C09095=1086.401,201.775,-73.711,175.633,21.629,153.454
C09096=1086.407,202.025,-73.734,175.636,21.631,153.454
C09097=1086.413,202.273,-73.758,175.638,21.633,153.454
C09098=1086.418,202.522,-73.781,175.641,21.634,153.454
C09099=1086.424,202.770,-73.805,175.644,21.636,153.454
C09100=1086.429,203.020,-73.828,175.647,21.638,153.453
C09101=1086.436,203.268,-73.852,175.649,21.640,153.454
C09102=1086.441,203.517,-73.876,175.652,21.641,153.453
C09103=1086.446,203.766,-73.900,175.654,21.643,153.453
C09104=1086.452,204.015,-73.923,175.657,21.644,153.453
C09105=1086.457,204.264,-73.947,175.659,21.646,153.453
C09106=1086.463,204.512,-73.971,175.663,21.648,153.453
C09107=1086.468,204.761,-73.995,175.665,21.650,153.453
C09108=1086.474,205.010,-74.019,175.668,21.651,153.453
C09109=1086.480,205.258,-74.042,175.670,21.653,153.453
C09110=1086.485,205.507,-74.066,175.673,21.654,153.453
C09111=1086.491,205.756,-74.090,175.675,21.656,153.453
C09112=1086.497,206.005,-74.114,175.679,21.658,153.453
C09113=1086.502,206.254,-74.138,175.681,21.660,153.453
C09114=1086.508,206.502,-74.161,175.684,21.661,153.453
C09115=1086.513,206.751,-74.186,175.686,21.663,153.453
C09116=1086.519,207.001,-74.210,175.689,21.665,153.453
C09117=1086.525,207.249,-74.233,175.692,21.666,153.453
C09118=1086.547,208.275,-74.332,175.771,21.707,153.449
C09119=1086.557,208.662,-74.370,175.775,21.711,153.449
C09120=1086.565,209.049,-74.408,175.779,21.715,153.450
C09121=1086.574,209.435,-74.446,175.782,21.719,153.450
C09122=1086.582,209.821,-74.484,175.787,21.723,153.450
C09123=1086.588,210.071,-74.509,175.789,21.726,153.450
C09124=1086.594,210.319,-74.532,175.792,21.728,153.450
C09125=1086.600,210.568,-74.557,175.795,21.731,153.451
C09126=1086.605,210.816,-74.582,175.797,21.733,153.451
C09127=1086.611,211.065,-74.606,175.800,21.736,153.451
C09128=1086.617,211.314,-74.631,175.802,21.738,153.451
C09129=1086.622,211.563,-74.655,175.805,21.741,153.451
C09130=1086.628,211.812,-74.680,175.807,21.744,153.451
C09131=1086.633,212.060,-74.705,175.810,21.747,153.452
C09132=1086.639,212.309,-74.729,175.813,21.749,153.452
C09133=1086.645,212.558,-74.754,175.815,21.752,153.452
C09134=1086.650,212.806,-74.779,175.818,21.754,153.452
C09135=1086.656,213.055,-74.803,175.820,21.757,153.452
C09136=1086.661,213.304,-74.827,175.823,21.760,153.452
C09137=1086.667,213.553,-74.852,175.825,21.762,153.453
C09138=1086.672,213.801,-74.878,175.829,21.765,153.453
C09139=1086.678,214.051,-74.902,175.831,21.767,153.453
C09140=1086.683,214.299,-74.926,175.833,21.770,153.453
C09141=1086.689,214.547,-74.951,175.836,21.772,153.453
C09142=1086.695,214.796,-74.976,175.838,21.775,153.453
C09143=1086.700,215.044,-75.001,175.841,21.778,153.454
C09144=1086.706,215.294,-75.026,175.843,21.780,153.454
C09145=1086.711,215.543,-75.051,175.847,21.783,153.454
C09146=1086.717,215.791,-75.076,175.849,21.786,153.454
C09147=1086.722,216.040,-75.100,175.852,21.788,153.454
C09148=1086.729,216.288,-75.125,175.854,21.791,153.454
C09149=1086.734,216.537,-75.150,175.856,21.793,153.454
C09150=1086.740,216.786,-75.175,175.859,21.796,153.455
C09151=1086.745,217.035,-75.200,175.862,21.798,153.455
C09152=1086.751,217.283,-75.225,175.865,21.801,153.455
C09153=1086.756,217.532,-75.249,175.867,21.804,153.455
C09154=1086.762,217.781,-75.275,175.870,21.806,153.455
C09155=1086.768,218.029,-75.299,175.872,21.809,153.456
C09156=1086.773,218.278,-75.325,175.875,21.812,153.456
C09157=1086.779,218.527,-75.350,175.877,21.814,153.456
C09158=1086.785,218.775,-75.375,175.881,21.817,153.456
C09159=1086.791,219.025,-75.399,175.883,21.820,153.456
C09160=1086.795,219.273,-75.425,175.886,21.822,153.456
C09161=1086.802,219.522,-75.450,175.888,21.825,153.456
C09162=1086.807,219.770,-75.474,175.891,21.828,153.457
C09163=1086.813,220.019,-75.500,175.893,21.830,153.457
C09164=1086.818,220.268,-75.525,175.896,21.832,153.457
C09165=1086.824,220.516,-75.550,175.899,21.835,153.457
C09166=1086.830,220.765,-75.575,175.901,21.837,153.457
C09167=1086.836,221.014,-75.600,175.904,21.840,153.457
C09168=1086.841,221.263,-75.625,175.906,21.843,153.457
C09169=1086.847,221.511,-75.651,175.909,21.845,153.458
C09170=1086.853,221.759,-75.676,175.912,21.848,153.458
C09171=1086.862,222.150,-75.715,175.916,21.852,153.458
C09172=1086.870,222.541,-75.755,175.920,21.856,153.458
C09173=1086.879,222.931,-75.794,175.925,21.861,153.459
C09174=1086.887,223.322,-75.835,175.928,21.865,153.459
C09175=1086.894,223.570,-75.860,175.931,21.868,153.459
C09176=1086.899,223.818,-75.885,175.934,21.870,153.459
C09177=1086.904,224.068,-75.910,175.937,21.873,153.459
C09178=1086.910,224.317,-75.936,175.939,21.875,153.460
C09179=1086.916,224.565,-75.961,175.942,21.878,153.460
C09180=1086.921,224.814,-75.987,175.944,21.880,153.460
C09181=1086.927,225.062,-76.012,175.947,21.883,153.460
C09182=1086.932,225.311,-76.038,175.950,21.885,153.460
C09183=1086.938,225.559,-76.063,175.952,21.889,153.460
C09184=1086.944,225.808,-76.089,175.955,21.891,153.461
C09185=1086.949,226.056,-76.114,175.958,21.894,153.461
C09186=1086.955,226.305,-76.140,175.960,21.896,153.461
C09187=1086.961,226.554,-76.165,175.963,21.899,153.461
C09188=1086.966,226.804,-76.191,175.965,21.901,153.461
C09189=1086.972,227.051,-76.216,175.968,21.904,153.461
C09190=1086.977,227.300,-76.241,175.972,21.907,153.461
C09191=1086.983,227.549,-76.267,175.974,21.909,153.462
C09192=1086.989,227.797,-76.293,175.977,21.912,153.462
C09193=1086.995,228.045,-76.318,175.979,21.915,153.462
C09194=1087.000,228.294,-76.344,175.982,21.917,153.462
C09195=1087.007,228.543,-76.370,175.985,21.920,153.462
C09196=1087.012,228.792,-76.396,175.987,21.923,153.462
C09197=1087.017,229.040,-76.421,175.990,21.925,153.463
C09198=1087.023,229.289,-76.446,175.993,21.928,153.463
C09199=1087.029,229.538,-76.472,175.995,21.931,153.463
C09200=1087.035,229.787,-76.498,175.998,21.933,153.463
C09201=1087.040,230.036,-76.524,176.000,21.936,153.463
C09202=1087.046,230.284,-76.549,176.003,21.939,153.463
C09203=1087.052,230.532,-76.575,176.006,21.941,153.464
C09204=1087.057,230.781,-76.601,176.009,21.944,153.464
C09205=1087.063,231.030,-76.627,176.012,21.947,153.464
C09206=1087.068,231.278,-76.652,176.014,21.949,153.464
C09207=1087.074,231.527,-76.678,176.017,21.952,153.464
C09208=1087.079,231.775,-76.705,176.019,21.955,153.464
C09209=1087.085,232.024,-76.731,176.022,21.957,153.465
C09210=1087.091,232.273,-76.756,176.025,21.960,153.465
C09211=1087.096,232.522,-76.782,176.028,21.963,153.465
C09212=1087.102,232.770,-76.808,176.030,21.965,153.465
C09213=1087.107,233.019,-76.834,176.033,21.968,153.465
C09214=1087.113,233.267,-76.859,176.036,21.971,153.465
C09215=1087.119,233.516,-76.886,176.038,21.973,153.466
C09216=1087.125,233.765,-76.912,176.041,21.976,153.466
C09217=1087.130,234.014,-76.938,176.044,21.978,153.466
C09218=1087.135,234.261,-76.964,176.047,21.981,153.466
C09219=1087.141,234.510,-76.990,176.049,21.984,153.466
C09220=1087.147,234.759,-77.016,176.052,21.986,153.466
C09221=1087.153,235.007,-77.042,176.055,21.990,153.467
C09222=1087.158,235.256,-77.068,176.057,21.992,153.467
C09223=1087.166,235.637,-77.108,176.062,21.996,153.467
C09224=1087.175,236.019,-77.149,176.066,22.000,153.467
C09225=1087.184,236.402,-77.188,176.070,22.005,153.468
C09226=1087.192,236.783,-77.228,176.074,22.009,153.468
C09227=1087.198,237.031,-77.255,176.077,22.011,153.468
C09228=1087.204,237.280,-77.281,176.079,22.014,153.468
C09229=1087.209,237.529,-77.307,176.082,22.017,153.468
C09230=1087.215,237.778,-77.333,176.085,22.019,153.469
C09231=1087.221,238.026,-77.360,176.088,22.022,153.469
C09232=1087.226,238.274,-77.387,176.091,22.025,153.469
C09233=1087.232,238.523,-77.413,176.093,22.027,153.469
C09234=1087.238,238.772,-77.439,176.096,22.030,153.469
C09235=1087.243,239.021,-77.465,176.098,22.032,153.469
C09236=1087.249,239.269,-77.492,176.101,22.036,153.470
C09237=1087.255,239.517,-77.519,176.104,22.038,153.470
C09238=1087.260,239.766,-77.544,176.107,22.041,153.470
C09239=1087.266,240.015,-77.571,176.110,22.044,153.470
C09240=1087.272,240.263,-77.598,176.112,22.046,153.470
C09241=1087.277,240.512,-77.624,176.115,22.049,153.470
C09242=1087.283,240.761,-77.650,176.118,22.052,153.471
C09243=1087.289,241.009,-77.677,176.120,22.054,153.471
C09244=1087.294,241.258,-77.703,176.124,22.057,153.471
C09245=1087.300,241.506,-77.730,176.127,22.060,153.471
C09246=1087.306,241.755,-77.756,176.129,22.062,153.471
C09247=1087.312,242.003,-77.783,176.132,22.065,153.471
C09248=1087.317,242.252,-77.809,176.134,22.068,153.472
C09249=1087.323,242.500,-77.835,176.137,22.070,153.472
C09250=1087.329,242.749,-77.862,176.140,22.074,153.472
C09251=1087.334,242.997,-77.889,176.143,22.076,153.472
C09252=1087.340,243.245,-77.915,176.146,22.079,153.472
C09253=1087.345,243.495,-77.942,176.148,22.081,153.473
C09254=1087.351,243.743,-77.969,176.151,22.084,153.473
C09255=1087.356,243.991,-77.995,176.154,22.087,153.473
C09256=1087.362,244.240,-78.022,176.156,22.090,153.473
C09257=1087.367,244.488,-78.049,176.159,22.092,153.473
C09258=1087.373,244.737,-78.076,176.162,22.095,153.473
C09259=1087.379,244.985,-78.102,176.164,22.098,153.474
C09260=1087.384,245.233,-78.129,176.168,22.101,153.474
C09261=1087.390,245.482,-78.156,176.171,22.104,153.474
C09262=1087.396,245.731,-78.183,176.173,22.106,153.474
C09263=1087.402,245.980,-78.210,176.176,22.109,153.474
C09264=1087.407,246.229,-78.236,176.179,22.112,153.475
C09265=1087.412,246.477,-78.263,176.181,22.114,153.475
C09266=1087.418,246.725,-78.290,176.184,22.117,153.475
C09267=1087.424,246.973,-78.317,176.187,22.119,153.475
C09268=1087.430,247.222,-78.344,176.190,22.123,153.475
C09269=1087.435,247.470,-78.371,176.193,22.125,153.476
C09270=1087.441,247.719,-78.398,176.195,22.128,153.476
C09271=1087.446,247.967,-78.425,176.198,22.131,153.476
C09272=1087.451,248.216,-78.452,176.201,22.134,153.476
C09273=1087.457,248.465,-78.479,176.203,22.136,153.476
C09274=1087.463,248.713,-78.506,176.206,22.139,153.476
C09275=1087.472,249.088,-78.547,176.211,22.144,153.477
C09276=1087.479,249.463,-78.587,176.215,22.147,153.477
C09277=1087.488,249.837,-78.628,176.219,22.152,153.477
C09278=1087.496,250.213,-78.669,176.223,22.156,153.478
C09279=1087.501,250.462,-78.696,176.226,22.159,153.478
C09280=1087.507,250.709,-78.724,176.229,22.162,153.478
C09281=1087.514,250.958,-78.751,176.231,22.164,153.478
C09282=1087.519,251.207,-78.778,176.234,22.168,153.478
C09283=1087.524,251.456,-78.805,176.237,22.170,153.479
C09284=1087.530,251.704,-78.832,176.240,22.173,153.479
C09285=1087.535,251.952,-78.860,176.243,22.176,153.479
C09286=1087.540,252.201,-78.886,176.246,22.179,153.479
C09287=1087.546,252.449,-78.915,176.248,22.181,153.479
C09288=1087.552,252.698,-78.941,176.251,22.184,153.480
C09289=1087.557,252.946,-78.969,176.254,22.187,153.480
C09290=1087.563,253.194,-78.996,176.256,22.189,153.480
C09291=1087.569,253.444,-79.024,176.259,22.192,153.480
C09292=1087.575,253.692,-79.050,176.262,22.196,153.480
C09293=1087.580,253.940,-79.078,176.266,22.198,153.481
C09294=1087.586,254.188,-79.105,176.268,22.201,153.481
C09295=1087.591,254.436,-79.133,176.271,22.204,153.481
C09296=1087.597,254.686,-79.160,176.274,22.207,153.481
C09297=1087.603,254.934,-79.187,176.276,22.209,153.481
C09298=1087.608,255.182,-79.215,176.279,22.212,153.482
C09299=1087.614,255.431,-79.242,176.282,22.215,153.482
C09300=1087.620,255.679,-79.270,176.284,22.217,153.482
C09301=1087.625,255.928,-79.297,176.288,22.220,153.482
C09302=1087.631,256.176,-79.325,176.291,22.224,153.482
C09303=1087.637,256.424,-79.353,176.294,22.226,153.483
C09304=1087.642,256.673,-79.380,176.296,22.229,153.483
C09305=1087.648,256.921,-79.407,176.299,22.232,153.483
C09306=1087.653,257.170,-79.435,176.302,22.235,153.483
C09307=1087.660,257.418,-79.462,176.304,22.237,153.483
C09308=1087.665,257.667,-79.490,176.307,22.240,153.483
C09309=1087.671,257.915,-79.517,176.310,22.243,153.484
C09310=1087.677,258.163,-79.545,176.313,22.246,153.484
C09311=1087.682,258.412,-79.573,176.316,22.248,153.484
C09312=1087.688,258.660,-79.600,176.319,22.251,153.484
C09313=1087.694,258.908,-79.628,176.322,22.254,153.484
C09314=1087.699,259.158,-79.656,176.325,22.257,153.485
C09315=1087.705,259.405,-79.683,176.327,22.259,153.485
C09316=1087.711,259.653,-79.711,176.330,22.263,153.485
C09317=1087.716,259.903,-79.739,176.333,22.265,153.485
C09318=1087.722,260.150,-79.766,176.336,22.268,153.485
C09319=1087.728,260.399,-79.795,176.339,22.271,153.486
C09320=1087.734,260.647,-79.823,176.342,22.274,153.486
C09321=1087.740,260.895,-79.850,176.345,22.277,153.486
C09322=1087.745,261.144,-79.877,176.347,22.279,153.486
C09323=1087.751,261.392,-79.905,176.350,22.282,153.486
C09324=1087.757,261.641,-79.934,176.353,22.285,153.487
C09325=1087.763,261.889,-79.961,176.356,22.288,153.487
C09326=1087.769,262.138,-79.989,176.358,22.290,153.487
C09327=1087.777,262.510,-80.031,176.363,22.295,153.487
C09328=1087.786,262.882,-80.073,176.368,22.299,153.487
C09329=1087.794,263.254,-80.115,176.371,22.303,153.488
C09330=1087.803,263.626,-80.156,176.376,22.307,153.488
C09331=1087.810,263.875,-80.184,176.379,22.310,153.488
C09332=1087.815,264.123,-80.212,176.381,22.312,153.488
C09333=1087.821,264.371,-80.240,176.384,22.316,153.489
C09334=1087.826,264.619,-80.268,176.388,22.318,153.489
C09335=1087.832,264.868,-80.297,176.390,22.322,153.489
C09336=1087.837,265.116,-80.325,176.394,22.324,153.489
C09337=1087.843,265.365,-80.353,176.396,22.327,153.490
C09338=1087.849,265.613,-80.381,176.399,22.330,153.490
C09339=1087.855,265.862,-80.409,176.402,22.333,153.490
C09340=1087.860,266.110,-80.437,176.405,22.336,153.490
C09341=1087.866,266.359,-80.466,176.407,22.338,153.490
C09342=1087.871,266.607,-80.493,176.410,22.342,153.491
C09343=1087.877,266.855,-80.521,176.413,22.344,153.491
C09344=1087.883,267.103,-80.550,176.416,22.348,153.491
C09345=1087.889,267.352,-80.579,176.419,22.350,153.491
C09346=1087.894,267.600,-80.607,176.421,22.353,153.492
C09347=1087.900,267.848,-80.635,176.425,22.356,153.492
C09348=1087.905,268.096,-80.663,176.428,22.359,153.492
C09349=1087.911,268.345,-80.691,176.431,22.362,153.492
C09350=1087.917,268.593,-80.720,176.433,22.364,153.492
C09351=1087.923,268.841,-80.748,176.436,22.368,153.493
C09352=1087.928,269.090,-80.777,176.439,22.370,153.493
C09353=1087.934,269.338,-80.805,176.442,22.374,153.493
C09354=1087.939,269.586,-80.834,176.445,22.377,153.493
C09355=1087.945,269.835,-80.862,176.447,22.379,153.493
C09356=1087.951,270.083,-80.891,176.450,22.382,153.494
C09357=1087.957,270.331,-80.919,176.453,22.385,153.494
C09358=1087.963,270.580,-80.948,176.456,22.388,153.494
C09359=1087.968,270.828,-80.976,176.459,22.391,153.494
C09360=1087.974,271.076,-81.005,176.463,22.394,153.495
C09361=1087.979,271.325,-81.033,176.465,22.397,153.495
C09362=1087.985,271.573,-81.061,176.468,22.400,153.495
C09363=1087.991,271.821,-81.090,176.471,22.403,153.495
C09364=1087.996,272.069,-81.118,176.474,22.406,153.495
C09365=1088.002,272.317,-81.148,176.477,22.409,153.496
C09366=1088.008,272.566,-81.176,176.479,22.411,153.496
C09367=1088.013,272.814,-81.204,176.482,22.415,153.496
C09368=1088.019,273.062,-81.233,176.485,22.417,153.496
C09369=1088.024,273.311,-81.262,176.488,22.421,153.497
C09370=1088.030,273.559,-81.291,176.491,22.423,153.497
C09371=1088.036,273.808,-81.319,176.494,22.427,153.497
C09372=1088.042,274.055,-81.348,176.497,22.429,153.497
C09373=1088.047,274.304,-81.377,176.500,22.432,153.498
C09374=1088.053,274.552,-81.406,176.502,22.435,153.498
C09375=1088.059,274.800,-81.435,176.506,22.438,153.498
C09376=1088.064,275.049,-81.464,176.509,22.441,153.498
C09377=1088.070,275.297,-81.493,176.512,22.444,153.498
C09378=1088.076,275.545,-81.521,176.514,22.447,153.499
C09379=1088.085,275.920,-81.564,176.518,22.452,153.499
C09380=1088.093,276.295,-81.608,176.523,22.456,153.499
C09381=1088.102,276.670,-81.652,176.527,22.461,153.500
C09382=1088.110,277.044,-81.696,176.532,22.466,153.500
C09383=1088.116,277.293,-81.724,176.534,22.468,153.500
C09384=1088.122,277.541,-81.754,176.537,22.471,153.501
C09385=1088.127,277.790,-81.783,176.540,22.474,153.501
C09386=1088.133,278.037,-81.812,176.543,22.477,153.501
C09387=1088.138,278.286,-81.841,176.546,22.480,153.501
C09388=1088.144,278.535,-81.870,176.549,22.483,153.502
C09389=1088.149,278.782,-81.899,176.552,22.486,153.502
C09390=1088.156,279.030,-81.928,176.554,22.489,153.502
C09391=1088.161,279.279,-81.958,176.558,22.492,153.502
C09392=1088.167,279.528,-81.986,176.561,22.495,153.503
C09393=1088.173,279.776,-82.016,176.564,22.498,153.503
C09394=1088.178,280.023,-82.044,176.567,22.501,153.503
C09395=1088.184,280.272,-82.074,176.570,22.504,153.503
C09396=1088.190,280.520,-82.103,176.573,22.508,153.504
C09397=1088.195,280.768,-82.133,176.576,22.510,153.504
C09398=1088.201,281.016,-82.161,176.578,22.513,153.504
C09399=1088.207,281.264,-82.191,176.581,22.516,153.504
C09400=1088.213,281.512,-82.220,176.584,22.519,153.505
C09401=1088.218,281.761,-82.250,176.587,22.523,153.505
C09402=1088.224,282.009,-82.279,176.590,22.526,153.505
C09403=1088.230,282.257,-82.308,176.593,22.529,153.505
C09404=1088.235,282.505,-82.338,176.596,22.532,153.506
C09405=1088.241,282.754,-82.367,176.599,22.535,153.506
C09406=1088.247,283.002,-82.396,176.602,22.538,153.506
C09407=1088.252,283.250,-82.426,176.604,22.541,153.506
C09408=1088.257,283.498,-82.455,176.607,22.544,153.507
C09409=1088.263,283.746,-82.484,176.610,22.547,153.507
C09410=1088.269,283.995,-82.514,176.613,22.550,153.507
C09411=1088.274,284.243,-82.543,176.616,22.554,153.507
C09412=1088.281,284.491,-82.573,176.619,22.557,153.508
C09413=1088.286,284.740,-82.602,176.622,22.560,153.508
C09414=1088.291,284.987,-82.631,176.625,22.563,153.508
C09415=1088.297,285.235,-82.662,176.628,22.566,153.508
C09416=1088.303,285.483,-82.691,176.631,22.569,153.509
C09417=1088.309,285.732,-82.720,176.634,22.572,153.509
C09418=1088.314,285.980,-82.750,176.636,22.575,153.509
C09419=1088.320,286.229,-82.780,176.639,22.578,153.510
C09420=1088.326,286.476,-82.809,176.642,22.581,153.510
C09421=1088.332,286.725,-82.839,176.645,22.585,153.510
C09422=1088.337,286.973,-82.869,176.649,22.587,153.510
C09423=1088.343,287.221,-82.898,176.652,22.591,153.511
C09424=1088.349,287.468,-82.928,176.655,22.594,153.511
C09425=1088.354,287.717,-82.957,176.657,22.597,153.511
C09426=1088.360,287.965,-82.987,176.660,22.600,153.511
C09427=1088.366,288.213,-83.017,176.664,22.603,153.512
C09428=1088.372,288.461,-83.046,176.667,22.606,153.512
C09429=1088.378,288.709,-83.077,176.670,22.609,153.512
C09430=1088.383,288.957,-83.106,176.673,22.613,153.512
C09431=1088.392,289.342,-83.152,176.677,22.617,153.513
C09432=1088.401,289.727,-83.199,176.681,22.622,153.513
C09433=1088.410,290.111,-83.245,176.686,22.627,153.514
C09434=1088.418,290.496,-83.292,176.690,22.632,153.514
C09435=1088.425,290.743,-83.321,176.693,22.635,153.515
C09436=1088.430,290.992,-83.351,176.696,22.639,153.515
C09437=1088.436,291.240,-83.381,176.699,22.642,153.515
C09438=1088.442,291.488,-83.411,176.703,22.645,153.515
C09439=1088.448,291.736,-83.441,176.705,22.648,153.516
C09440=1088.453,291.984,-83.471,176.708,22.651,153.516
C09441=1088.459,292.232,-83.501,176.711,22.654,153.516
C09442=1088.465,292.480,-83.532,176.714,22.657,153.516
C09443=1088.470,292.728,-83.561,176.717,22.661,153.517
C09444=1088.476,292.976,-83.592,176.720,22.664,153.517
C09445=1088.482,293.224,-83.622,176.723,22.667,153.517
C09446=1088.487,293.472,-83.652,176.726,22.670,153.518
C09447=1088.492,293.721,-83.683,176.729,22.674,153.518
C09448=1088.498,293.968,-83.713,176.732,22.677,153.518
C09449=1088.504,294.217,-83.743,176.734,22.680,153.519
C09450=1088.510,294.465,-83.773,176.737,22.683,153.519
C09451=1088.515,294.712,-83.803,176.740,22.686,153.519
C09452=1088.521,294.961,-83.833,176.743,22.689,153.519
C09453=1088.527,295.209,-83.863,176.746,22.693,153.520
C09454=1088.533,295.457,-83.894,176.749,22.696,153.520
C09455=1088.539,295.705,-83.924,176.752,22.699,153.520
C09456=1088.545,295.953,-83.955,176.755,22.702,153.521
C09457=1088.550,296.201,-83.984,176.758,22.705,153.521
C09458=1088.555,296.449,-84.015,176.761,22.709,153.521
C09459=1088.561,296.697,-84.046,176.764,22.712,153.522
C09460=1088.567,296.945,-84.076,176.767,22.716,153.522
C09461=1088.573,297.193,-84.106,176.770,22.719,153.522
C09462=1088.579,297.441,-84.137,176.773,22.722,153.522
C09463=1088.585,297.689,-84.167,176.776,22.725,153.523
C09464=1088.590,297.938,-84.198,176.779,22.728,153.523
C09465=1088.596,298.186,-84.228,176.782,22.732,153.523
C09466=1088.601,298.434,-84.258,176.785,22.735,153.524
C09467=1088.607,298.682,-84.289,176.789,22.739,153.524
C09468=1088.612,298.930,-84.320,176.792,22.742,153.524
C09469=1088.618,299.177,-84.350,176.795,22.746,153.525
C09470=1088.623,299.426,-84.381,176.797,22.749,153.525
C09471=1088.629,299.673,-84.411,176.800,22.752,153.525
C09472=1088.634,299.922,-84.442,176.803,22.756,153.526
C09473=1088.641,300.170,-84.473,176.806,22.759,153.526
C09474=1088.646,300.418,-84.504,176.809,22.763,153.526
C09475=1088.652,300.665,-84.535,176.812,22.766,153.527
C09476=1088.658,300.913,-84.565,176.815,22.769,153.527
C09477=1088.663,301.161,-84.596,176.818,22.773,153.527
C09478=1088.668,301.409,-84.627,176.821,22.776,153.528
C09479=1088.674,301.657,-84.658,176.824,22.779,153.528
C09480=1088.680,301.906,-84.688,176.827,22.783,153.528
C09481=1088.685,302.154,-84.719,176.830,22.786,153.529
C09482=1088.691,302.401,-84.750,176.833,22.789,153.529
C09483=1088.700,302.800,-84.800,176.838,22.795,153.530
C09484=1088.709,303.198,-84.849,176.842,22.800,153.530
C09485=1088.718,303.597,-84.899,176.848,22.806,153.531
C09486=1088.727,303.995,-84.949,176.852,22.811,153.531
C09487=1088.733,304.243,-84.979,176.855,22.815,153.532
C09488=1088.739,304.492,-85.011,176.858,22.818,153.532
C09489=1088.745,304.739,-85.042,176.861,22.822,153.532
C09490=1088.750,304.987,-85.073,176.864,22.825,153.533
C09491=1088.756,305.235,-85.103,176.867,22.829,153.533
C09492=1088.762,305.483,-85.135,176.870,22.832,153.533
C09493=1088.767,305.731,-85.166,176.873,22.835,153.534
C09494=1088.773,305.979,-85.196,176.876,22.839,153.534
C09495=1088.779,306.227,-85.229,176.879,22.842,153.534
C09496=1088.784,306.475,-85.259,176.882,22.846,153.535
C09497=1088.790,306.723,-85.291,176.885,22.849,153.535
C09498=1088.796,306.971,-85.321,176.888,22.852,153.535
C09499=1088.802,307.219,-85.353,176.891,22.856,153.536
C09500=1088.807,307.467,-85.383,176.894,22.859,153.536
C09501=1088.813,307.715,-85.415,176.897,22.863,153.537
C09502=1088.818,307.963,-85.446,176.900,22.867,153.537
C09503=1088.825,308.210,-85.477,176.903,22.870,153.537
C09504=1088.830,308.459,-85.509,176.906,22.873,153.538
C09505=1088.836,308.706,-85.540,176.909,22.877,153.538
C09506=1088.842,308.955,-85.571,176.912,22.880,153.538
C09507=1088.847,309.203,-85.603,176.915,22.884,153.539
C09508=1088.854,309.450,-85.634,176.918,22.887,153.539
C09509=1088.859,309.699,-85.665,176.921,22.890,153.539
C09510=1088.865,309.946,-85.697,176.924,22.894,153.540
C09511=1088.871,310.194,-85.728,176.928,22.898,153.540
C09512=1088.876,310.442,-85.759,176.930,22.901,153.540
C09513=1088.882,310.690,-85.791,176.933,22.905,153.541
C09514=1088.889,310.938,-85.822,176.936,22.908,153.541
C09515=1088.894,311.186,-85.853,176.939,22.912,153.542
C09516=1088.900,311.434,-85.885,176.942,22.915,153.542
C09517=1088.906,311.682,-85.917,176.945,22.918,153.542
C09518=1088.912,311.929,-85.948,176.948,22.922,153.543
C09519=1088.917,312.178,-85.980,176.951,22.925,153.543
C09520=1088.923,312.425,-86.011,176.955,22.929,153.543
C09521=1088.929,312.674,-86.043,176.958,22.933,153.544
C09522=1088.935,312.921,-86.074,176.960,22.936,153.544
C09523=1088.942,313.169,-86.106,176.964,22.940,153.544
C09524=1088.947,313.416,-86.137,176.966,22.943,153.545
C09525=1088.953,313.665,-86.169,176.969,22.946,153.545
C09526=1088.958,313.913,-86.200,176.972,22.950,153.546
C09527=1088.965,314.161,-86.232,176.976,22.954,153.546
C09528=1088.971,314.409,-86.264,176.979,22.957,153.546
C09529=1088.976,314.656,-86.295,176.982,22.961,153.547
C09530=1088.982,314.905,-86.327,176.985,22.964,153.547
C09531=1088.988,315.152,-86.359,176.988,22.968,153.547
C09532=1088.993,315.400,-86.391,176.990,22.972,153.548
C09533=1088.999,315.648,-86.423,176.993,22.975,153.548
C09534=1089.005,315.896,-86.455,176.997,22.979,153.549
C09535=1089.014,316.297,-86.507,177.001,22.985,153.549
C09536=1089.023,316.698,-86.558,177.006,22.991,153.550
C09537=1089.032,317.100,-86.610,177.011,22.997,153.551
C09538=1089.041,317.501,-86.662,177.016,23.003,153.551
C09539=1089.047,317.749,-86.693,177.019,23.007,153.552
C09540=1089.053,317.997,-86.725,177.022,23.011,153.552
C09541=1089.058,318.244,-86.757,177.025,23.014,153.553
C09542=1089.064,318.493,-86.789,177.028,23.018,153.553
C09543=1089.069,318.741,-86.822,177.031,23.022,153.554
C09544=1089.075,318.988,-86.854,177.034,23.026,153.554
C09545=1089.081,319.236,-86.886,177.037,23.029,153.554
C09546=1089.086,319.484,-86.918,177.040,23.033,153.555
C09547=1089.092,319.732,-86.950,177.043,23.037,153.555
C09548=1089.098,319.980,-86.983,177.046,23.040,153.556
C09549=1089.103,320.227,-87.015,177.049,23.044,153.556
C09550=1089.109,320.476,-87.047,177.052,23.048,153.557
C09551=1089.115,320.724,-87.079,177.055,23.052,153.557
C09552=1089.121,320.971,-87.111,177.058,23.055,153.558
C09553=1089.126,321.219,-87.144,177.061,23.059,153.558
C09554=1089.132,321.467,-87.176,177.064,23.063,153.558
C09555=1089.138,321.714,-87.208,177.067,23.067,153.559
C09556=1089.144,321.963,-87.240,177.070,23.071,153.559
C09557=1089.149,322.210,-87.274,177.073,23.074,153.560
C09558=1089.155,322.458,-87.305,177.076,23.078,153.560
C09559=1089.161,322.706,-87.337,177.080,23.082,153.561
C09560=1089.167,322.954,-87.370,177.082,23.086,153.561
C09561=1089.172,323.202,-87.403,177.085,23.089,153.561
C09562=1089.178,323.449,-87.435,177.088,23.093,153.562
C09563=1089.184,323.697,-87.467,177.092,23.098,153.562
C09564=1089.189,323.945,-87.500,177.095,23.101,153.563
C09565=1089.195,324.194,-87.532,177.097,23.105,153.563
C09566=1089.201,324.440,-87.565,177.100,23.109,153.564
C09567=1089.207,324.689,-87.597,177.103,23.112,153.564
C09568=1089.213,324.937,-87.630,177.107,23.116,153.565
C09569=1089.219,325.185,-87.662,177.109,23.120,153.565
C09570=1089.225,325.432,-87.695,177.112,23.124,153.566
C09571=1089.230,325.680,-87.727,177.115,23.128,153.566
C09572=1089.236,325.928,-87.760,177.119,23.132,153.566
C09573=1089.242,326.175,-87.793,177.122,23.136,153.567
C09574=1089.247,326.424,-87.825,177.124,23.140,153.567
C09575=1089.254,326.671,-87.858,177.127,23.143,153.568
C09576=1089.260,326.919,-87.891,177.131,23.147,153.568
C09577=1089.265,327.167,-87.923,177.134,23.151,153.569
C09578=1089.271,327.414,-87.956,177.137,23.155,153.569
C09579=1089.276,327.662,-87.989,177.139,23.159,153.570
C09580=1089.283,327.910,-88.022,177.143,23.163,153.570
C09581=1089.289,328.158,-88.054,177.146,23.167,153.571
C09582=1089.294,328.406,-88.087,177.149,23.170,153.571
C09583=1089.301,328.654,-88.120,177.152,23.175,153.572
C09584=1089.306,328.902,-88.153,177.155,23.178,153.572
C09585=1089.312,329.149,-88.186,177.158,23.182,153.572
C09586=1089.318,329.397,-88.218,177.161,23.186,153.573
C09587=1089.327,329.791,-88.271,177.166,23.193,153.574
C09588=1089.337,330.186,-88.323,177.171,23.199,153.574
C09589=1089.346,330.580,-88.376,177.176,23.205,153.575
C09590=1089.356,330.975,-88.428,177.181,23.211,153.576
C09591=1089.362,331.223,-88.461,177.184,23.215,153.577
C09592=1089.368,331.470,-88.494,177.186,23.219,153.577
C09593=1089.373,331.718,-88.527,177.190,23.223,153.577
C09594=1089.380,331.966,-88.560,177.193,23.227,153.578
C09595=1089.385,332.214,-88.593,177.196,23.231,153.578
C09596=1089.391,332.461,-88.627,177.199,23.235,153.579
C09597=1089.397,332.709,-88.659,177.202,23.240,153.580
C09598=1089.403,332.957,-88.693,177.205,23.243,153.580
C09599=1089.408,333.205,-88.726,177.208,23.248,153.581
C09600=1089.414,333.453,-88.760,177.211,23.252,153.581
C09601=1089.419,333.700,-88.792,177.214,23.256,153.582
C09602=1089.425,333.948,-88.825,177.218,23.260,153.582
C09603=1089.431,334.195,-88.859,177.220,23.264,153.583
C09604=1089.437,334.442,-88.892,177.223,23.268,153.583
C09605=1089.443,334.690,-88.925,177.227,23.272,153.584
C09606=1089.448,334.938,-88.959,177.229,23.277,153.584
C09607=1089.454,335.187,-88.992,177.232,23.281,153.585
C09608=1089.460,335.434,-89.026,177.236,23.285,153.585
C09609=1089.467,335.682,-89.059,177.239,23.289,153.586
C09610=1089.472,335.930,-89.093,177.242,23.293,153.586
C09611=1089.478,336.177,-89.126,177.245,23.297,153.587
C09612=1089.484,336.425,-89.160,177.248,23.302,153.588
C09613=1089.489,336.673,-89.193,177.251,23.306,153.588
C09614=1089.495,336.920,-89.226,177.254,23.310,153.589
C09615=1089.501,337.168,-89.260,177.257,23.314,153.589
C09616=1089.507,337.415,-89.293,177.260,23.318,153.590
C09617=1089.512,337.663,-89.327,177.263,23.323,153.590
C09618=1089.518,337.911,-89.361,177.267,23.327,153.591
C09619=1089.524,338.159,-89.394,177.269,23.331,153.591
C09620=1089.531,338.406,-89.428,177.272,23.335,153.592
C09621=1089.537,338.654,-89.461,177.276,23.339,153.592
C09622=1089.542,338.902,-89.495,177.278,23.343,153.593
C09623=1089.548,339.149,-89.529,177.282,23.348,153.593
C09624=1089.554,339.397,-89.562,177.285,23.352,153.594
C09625=1089.559,339.645,-89.596,177.287,23.357,153.595
C09626=1089.565,339.892,-89.629,177.291,23.361,153.595
C09627=1089.571,340.140,-89.663,177.294,23.365,153.596
C09628=1089.577,340.387,-89.698,177.297,23.370,153.596
C09629=1089.583,340.636,-89.731,177.300,23.374,153.597
C09630=1089.589,340.883,-89.765,177.303,23.378,153.598
C09631=1089.594,341.131,-89.799,177.306,23.383,153.598
C09632=1089.600,341.378,-89.833,177.309,23.387,153.599
C09633=1089.605,341.626,-89.867,177.312,23.391,153.599
C09634=1089.611,341.874,-89.901,177.315,23.396,153.600
C09635=1089.617,342.122,-89.935,177.319,23.400,153.601
C09636=1089.623,342.369,-89.969,177.321,23.404,153.601
C09637=1089.629,342.617,-90.002,177.325,23.409,153.602
C09638=1089.635,342.864,-90.036,177.328,23.413,153.602
C09639=1089.644,343.253,-90.090,177.332,23.420,153.603
C09640=1089.653,343.641,-90.143,177.337,23.427,153.604
C09641=1089.662,344.030,-90.197,177.342,23.434,153.605
C09642=1089.671,344.419,-90.251,177.347,23.441,153.606
C09643=1089.677,344.666,-90.285,177.349,23.445,153.607
C09644=1089.683,344.913,-90.319,177.353,23.450,153.607
C09645=1089.689,345.161,-90.353,177.356,23.454,153.608
C09646=1089.695,345.409,-90.386,177.359,23.459,153.609
C09647=1089.700,345.657,-90.421,177.362,23.463,153.609
C09648=1089.706,345.904,-90.455,177.365,23.468,153.610
C09649=1089.712,346.152,-90.490,177.368,23.472,153.610
C09650=1089.718,346.399,-90.524,177.371,23.477,153.611
C09651=1089.723,346.647,-90.558,177.374,23.481,153.612
C09652=1089.729,346.894,-90.592,177.378,23.486,153.612
C09653=1089.736,347.142,-90.627,177.380,23.491,153.613
C09654=1089.741,347.390,-90.661,177.384,23.495,153.614
C09655=1089.747,347.637,-90.695,177.386,23.500,153.614
C09656=1089.753,347.885,-90.730,177.390,23.504,153.615
C09657=1089.758,348.132,-90.765,177.393,23.509,153.616
C09658=1089.765,348.379,-90.799,177.396,23.514,153.616
C09659=1089.771,348.627,-90.834,177.399,23.518,153.617
C09660=1089.776,348.875,-90.868,177.402,23.523,153.618
C09661=1089.782,349.122,-90.902,177.405,23.527,153.618
C09662=1089.788,349.370,-90.937,177.408,23.532,153.619
C09663=1089.794,349.618,-90.971,177.411,23.537,153.620
C09664=1089.800,349.864,-91.006,177.414,23.542,153.620
C09665=1089.805,350.113,-91.041,177.417,23.546,153.621
C09666=1089.811,350.360,-91.075,177.421,23.551,153.622
C09667=1089.818,350.608,-91.110,177.424,23.556,153.622
C09668=1089.823,350.855,-91.145,177.427,23.560,153.623
C09669=1089.829,351.102,-91.179,177.430,23.565,153.624
C09670=1089.835,351.350,-91.214,177.433,23.570,153.624
C09671=1089.841,351.598,-91.248,177.436,23.575,153.625
C09672=1089.847,351.845,-91.284,177.439,23.579,153.626
C09673=1089.853,352.093,-91.318,177.442,23.584,153.626
C09674=1089.858,352.340,-91.353,177.445,23.588,153.627
C09675=1089.864,352.588,-91.388,177.448,23.593,153.628
C09676=1089.870,352.835,-91.422,177.452,23.598,153.628
C09677=1089.876,353.083,-91.458,177.454,23.603,153.629
C09678=1089.881,353.330,-91.492,177.458,23.608,153.630
C09679=1089.888,353.577,-91.527,177.460,23.612,153.631
C09680=1089.893,353.825,-91.562,177.464,23.617,153.631
C09681=1089.900,354.072,-91.597,177.466,23.622,153.632
C09682=1089.905,354.320,-91.632,177.470,23.627,153.633
C09683=1089.911,354.568,-91.667,177.473,23.632,153.633
C09684=1089.917,354.815,-91.702,177.476,23.637,153.634
C09685=1089.923,355.062,-91.737,177.479,23.642,153.635
C09686=1089.928,355.310,-91.772,177.482,23.646,153.636
C09687=1089.934,355.557,-91.807,177.485,23.651,153.636
C09688=1089.940,355.805,-91.842,177.488,23.657,153.637
C09689=1089.946,356.052,-91.877,177.491,23.661,153.638
C09690=1089.952,356.300,-91.912,177.494,23.666,153.638
C09691=1089.961,356.691,-91.968,177.499,23.674,153.640
C09692=1089.971,357.083,-92.024,177.504,23.681,153.641
C09693=1089.980,357.473,-92.080,177.509,23.690,153.642
C09694=1089.990,357.864,-92.135,177.514,23.697,153.643
C09695=1089.995,358.111,-92.170,177.517,23.703,153.644
C09696=1090.001,358.360,-92.205,177.520,23.707,153.645
C09697=1090.006,358.607,-92.241,177.523,23.713,153.646
C09698=1090.013,358.854,-92.276,177.526,23.718,153.646
C09699=1090.019,359.102,-92.312,177.529,23.723,153.647
C09700=1090.025,359.349,-92.347,177.532,23.728,153.648
C09701=1090.031,359.596,-92.383,177.536,23.733,153.649
C09702=1090.037,359.843,-92.418,177.538,23.737,153.649
C09703=1090.043,360.091,-92.453,177.542,23.743,153.650
C09704=1090.049,360.339,-92.488,177.545,23.748,153.651
C09705=1090.054,360.586,-92.524,177.547,23.753,153.652
C09706=1090.060,360.834,-92.559,177.551,23.758,153.653
C09707=1090.065,361.081,-92.595,177.554,23.764,153.653
C09708=1090.071,361.328,-92.630,177.557,23.768,153.654
C09709=1090.078,361.575,-92.667,177.560,23.774,153.655
C09710=1090.083,361.822,-92.702,177.563,23.779,153.656
C09711=1090.090,362.070,-92.737,177.566,23.784,153.657
C09712=1090.096,362.317,-92.773,177.569,23.789,153.657
C09713=1090.101,362.564,-92.809,177.573,23.794,153.658
C09714=1090.108,362.812,-92.844,177.575,23.799,153.659
C09715=1090.114,363.060,-92.880,177.578,23.805,153.660
C09716=1090.119,363.307,-92.915,177.582,23.810,153.661
C09717=1090.125,363.554,-92.952,177.585,23.816,153.661
C09718=1090.131,363.801,-92.988,177.587,23.821,153.662
C09719=1090.137,364.049,-93.023,177.591,23.826,153.663
C09720=1090.143,364.296,-93.059,177.594,23.831,153.664
C09721=1090.149,364.544,-93.094,177.596,23.836,153.665
C09722=1090.155,364.791,-93.131,177.600,23.842,153.666
C09723=1090.161,365.038,-93.166,177.603,23.847,153.666
C09724=1090.167,365.285,-93.202,177.606,23.853,153.667
C09725=1090.173,365.533,-93.238,177.609,23.857,153.668
C09726=1090.179,365.780,-93.274,177.612,23.863,153.669
C09727=1090.184,366.027,-93.310,177.616,23.868,153.670
C09728=1090.190,366.275,-93.346,177.619,23.874,153.671
C09729=1090.196,366.522,-93.382,177.621,23.879,153.672
C09730=1090.202,366.769,-93.419,177.625,23.885,153.672
C09731=1090.208,367.016,-93.454,177.628,23.890,153.673
C09732=1090.213,367.264,-93.491,177.631,23.896,153.674
C09733=1090.219,367.511,-93.527,177.634,23.901,153.675
C09734=1090.225,367.759,-93.562,177.637,23.907,153.676
C09735=1090.231,368.005,-93.599,177.640,23.912,153.677
C09736=1090.238,368.252,-93.635,177.643,23.918,153.678
C09737=1090.243,368.500,-93.671,177.646,23.923,153.679
C09738=1090.249,368.747,-93.708,177.649,23.929,153.680
C09739=1090.255,368.995,-93.744,177.652,23.934,153.680
C09740=1090.260,369.242,-93.780,177.655,23.940,153.681
C09741=1090.267,369.489,-93.817,177.658,23.945,153.682
C09742=1090.273,369.736,-93.852,177.661,23.951,153.683
C09743=1090.282,370.143,-93.912,177.666,23.960,153.685
C09744=1090.291,370.550,-93.972,177.671,23.969,153.686
C09745=1090.302,370.956,-94.032,177.676,23.979,153.688
C09746=1090.312,371.363,-94.092,177.682,23.988,153.689
C09747=1090.318,371.610,-94.128,177.685,23.993,153.690
C09748=1090.323,371.858,-94.165,177.688,23.999,153.691
C09749=1090.330,372.105,-94.201,177.690,24.005,153.692
C09750=1090.336,372.352,-94.238,177.694,24.011,153.693
C09751=1090.342,372.599,-94.275,177.697,24.016,153.694
C09752=1090.348,372.846,-94.311,177.700,24.022,153.695
C09753=1090.354,373.093,-94.347,177.703,24.028,153.696
C09754=1090.359,373.340,-94.384,177.707,24.033,153.697
C09755=1090.366,373.587,-94.421,177.709,24.039,153.698
C09756=1090.371,373.835,-94.457,177.712,24.045,153.699
C09757=1090.377,374.082,-94.493,177.715,24.051,153.700
C09758=1090.383,374.330,-94.531,177.719,24.056,153.701
C09759=1090.389,374.577,-94.567,177.722,24.062,153.702
C09760=1090.395,374.824,-94.604,177.725,24.068,153.703
C09761=1090.402,375.070,-94.641,177.728,24.074,153.704
C09762=1090.407,375.318,-94.678,177.730,24.080,153.705
C09763=1090.414,375.565,-94.715,177.733,24.086,153.706
C09764=1090.419,375.812,-94.752,177.737,24.092,153.707
C09765=1090.425,376.060,-94.789,177.740,24.098,153.708
C09766=1090.431,376.307,-94.825,177.743,24.104,153.709
C09767=1090.437,376.554,-94.862,177.746,24.110,153.710
C09768=1090.443,376.801,-94.899,177.749,24.116,153.711
C09769=1090.449,377.048,-94.936,177.752,24.122,153.712
C09770=1090.454,377.295,-94.973,177.756,24.128,153.713
C09771=1090.461,377.542,-95.010,177.758,24.134,153.714
C09772=1090.466,377.790,-95.047,177.761,24.139,153.715
C09773=1090.472,378.036,-95.085,177.764,24.146,153.716
C09774=1090.479,378.283,-95.121,177.767,24.152,153.717
C09775=1090.484,378.531,-95.158,177.770,24.158,153.718
C09776=1090.490,378.777,-95.196,177.774,24.164,153.719
C09777=1090.497,379.025,-95.232,177.777,24.170,153.720
C09778=1090.502,379.272,-95.269,177.780,24.176,153.721
C09779=1090.508,379.519,-95.307,177.783,24.182,153.722
C09780=1090.514,379.766,-95.344,177.786,24.189,153.723
C09781=1090.521,380.013,-95.382,177.789,24.195,153.724
C09782=1090.526,380.261,-95.419,177.792,24.201,153.725
C09783=1090.533,380.507,-95.456,177.795,24.207,153.726
C09784=1090.539,380.754,-95.493,177.799,24.213,153.728
C09785=1090.545,381.001,-95.531,177.802,24.220,153.729
C09786=1090.550,381.248,-95.568,177.805,24.226,153.730
C09787=1090.557,381.495,-95.605,177.808,24.232,153.731
C09788=1090.563,381.743,-95.642,177.810,24.238,153.732
C09789=1090.569,381.990,-95.680,177.813,24.244,153.733
C09790=1090.575,382.236,-95.718,177.816,24.251,153.734
C09791=1090.581,382.483,-95.754,177.819,24.257,153.735
C09792=1090.587,382.730,-95.792,177.822,24.263,153.736
C09793=1090.593,382.977,-95.830,177.825,24.269,153.737
C09794=1090.599,383.225,-95.867,177.828,24.276,153.739
C09795=1090.606,383.555,-95.918,177.833,24.285,153.740
C09796=1090.614,383.885,-95.968,177.837,24.294,153.742
C09797=1090.623,384.216,-96.018,177.842,24.302,153.743
C09798=1090.630,384.546,-96.069,177.845,24.311,153.745
C09799=1090.637,384.794,-96.106,177.848,24.317,153.746
C09800=1090.643,385.041,-96.144,177.851,24.323,153.747
C09801=1090.648,385.288,-96.182,177.854,24.330,153.748
C09802=1090.654,385.534,-96.220,177.857,24.336,153.749
C09803=1090.660,385.781,-96.257,177.861,24.344,153.751
C09804=1090.667,386.029,-96.295,177.864,24.350,153.752
C09805=1090.673,386.275,-96.333,177.867,24.357,153.753
C09806=1090.679,386.522,-96.371,177.870,24.363,153.754
C09807=1090.685,386.769,-96.409,177.873,24.370,153.755
C09808=1090.691,387.016,-96.447,177.876,24.377,153.757
C09809=1090.697,387.263,-96.485,177.879,24.383,153.758
C09810=1090.703,387.510,-96.522,177.882,24.390,153.759
C09811=1090.709,387.756,-96.560,177.885,24.396,153.760
C09812=1090.715,388.004,-96.599,177.888,24.403,153.761
C09813=1090.720,388.251,-96.637,177.891,24.410,153.763
C09814=1090.726,388.498,-96.674,177.894,24.416,153.764
C09815=1090.733,388.745,-96.712,177.898,24.424,153.765
C09816=1090.739,388.992,-96.750,177.901,24.430,153.766
C09817=1090.745,389.238,-96.789,177.904,24.437,153.767
C09818=1090.751,389.485,-96.827,177.907,24.444,153.769
C09819=1090.757,389.732,-96.865,177.910,24.450,153.770
C09820=1090.764,389.980,-96.903,177.913,24.457,153.771
C09821=1090.769,390.226,-96.942,177.916,24.464,153.773
C09822=1090.775,390.473,-96.980,177.919,24.471,153.774
C09823=1090.784,390.824,-97.033,177.924,24.481,153.776
C09824=1090.793,391.174,-97.088,177.928,24.490,153.777
C09825=1090.802,391.526,-97.143,177.932,24.500,153.779
C09826=1090.811,391.876,-97.197,177.937,24.511,153.781
C09827=1090.817,392.123,-97.235,177.940,24.517,153.782
C09828=1090.823,392.370,-97.274,177.943,24.524,153.784
C09829=1090.829,392.617,-97.312,177.945,24.531,153.785
C09830=1090.834,392.863,-97.351,177.948,24.539,153.786
C09831=1090.841,393.111,-97.389,177.952,24.546,153.787
C09832=1090.847,393.357,-97.428,177.955,24.553,153.789
C09833=1090.853,393.605,-97.466,177.958,24.560,153.790
C09834=1090.859,393.851,-97.505,177.961,24.567,153.792
C09835=1090.866,394.098,-97.543,177.964,24.574,153.793
C09836=1090.871,394.345,-97.582,177.967,24.582,153.794
C09837=1090.878,394.592,-97.620,177.970,24.589,153.796
C09838=1090.884,394.839,-97.660,177.973,24.596,153.797
C09839=1090.890,395.085,-97.698,177.976,24.603,153.798
C09840=1090.896,395.333,-97.737,177.979,24.610,153.800
C09841=1090.902,395.579,-97.775,177.983,24.618,153.801
C09842=1090.908,395.826,-97.815,177.986,24.625,153.802
C09843=1090.914,396.073,-97.852,177.988,24.633,153.804
C09844=1090.920,396.320,-97.892,177.991,24.640,153.805
C09845=1090.926,396.566,-97.930,177.994,24.647,153.807
C09846=1090.932,396.813,-97.970,177.998,24.655,153.808
C09847=1090.937,397.038,-98.005,178.001,24.661,153.809
C09848=1090.943,397.261,-98.040,178.003,24.668,153.811
C09849=1090.949,397.485,-98.076,178.006,24.675,153.812
C09850=1090.954,397.708,-98.111,178.009,24.681,153.813
C09851=1090.960,397.933,-98.146,178.012,24.689,153.814
C09852=1090.965,398.156,-98.181,178.014,24.695,153.816
C09853=1090.971,398.381,-98.216,178.017,24.702,153.817
C09854=1090.976,398.604,-98.252,178.020,24.709,153.818
C09855=1090.983,398.851,-98.291,178.023,24.716,153.820
C09856=1090.989,399.098,-98.330,178.026,24.724,153.821
C09857=1090.995,399.345,-98.370,178.029,24.732,153.823
C09858=1091.001,399.591,-98.408,178.032,24.739,153.824
C09859=1091.007,399.838,-98.448,178.034,24.747,153.826
C09860=1091.013,400.085,-98.487,178.038,24.755,153.827
C09861=1091.019,400.332,-98.526,178.041,24.762,153.829
C09862=1091.025,400.579,-98.565,178.044,24.770,153.830
C09863=1091.031,400.826,-98.604,178.047,24.778,153.832
C09864=1091.038,401.073,-98.644,178.050,24.785,153.833
C09865=1091.043,401.319,-98.683,178.054,24.793,153.835
C09866=1091.049,401.566,-98.723,178.056,24.801,153.836
C09867=1091.056,401.813,-98.762,178.059,24.809,153.838
C09868=1091.062,402.060,-98.801,178.063,24.817,153.839
C09869=1091.068,402.306,-98.840,178.066,24.825,153.841
C09870=1091.074,402.553,-98.880,178.068,24.833,153.842
C09871=1091.080,402.800,-98.920,178.072,24.841,153.844
C09872=1091.086,403.047,-98.959,178.075,24.848,153.845
C09873=1091.093,403.294,-98.998,178.078,24.857,153.847
C09874=1091.099,403.540,-99.038,178.081,24.864,153.848
C09875=1091.105,403.787,-99.077,178.084,24.872,153.850
C09876=1091.111,404.034,-99.117,178.087,24.881,153.852
C09877=1091.117,404.280,-99.157,178.090,24.889,153.853
C09878=1091.123,404.527,-99.197,178.094,24.897,153.855
C09879=1091.130,404.774,-99.237,178.096,24.905,153.856
C09880=1091.136,405.021,-99.276,178.100,24.913,153.858
C09881=1091.142,405.268,-99.316,178.102,24.921,153.860
C09882=1091.148,405.515,-99.356,178.106,24.930,153.861
C09883=1091.155,405.761,-99.396,178.109,24.938,153.863
C09884=1091.160,406.008,-99.435,178.112,24.946,153.865
C09885=1091.167,406.254,-99.475,178.115,24.954,153.866
C09886=1091.173,406.501,-99.514,178.118,24.963,153.868
C09887=1091.179,406.748,-99.555,178.121,24.971,153.869
C09888=1091.185,406.994,-99.595,178.125,24.980,153.871
C09889=1091.192,407.242,-99.634,178.127,24.988,153.873
C09890=1091.198,407.488,-99.674,178.131,24.996,153.874
C09891=1091.204,407.735,-99.715,178.133,25.004,153.876
C09892=1091.210,407.982,-99.755,178.137,25.013,153.878
C09893=1091.216,408.229,-99.795,178.139,25.022,153.880
C09894=1091.222,408.475,-99.835,178.143,25.030,153.881
C09895=1091.229,408.722,-99.875,178.146,25.038,153.883
C09896=1091.234,408.968,-99.916,178.149,25.047,153.885
C09897=1091.240,409.216,-99.955,178.152,25.056,153.886
C09898=1091.247,409.462,-99.995,178.155,25.065,153.888
C09899=1091.253,409.709,-100.036,178.159,25.073,153.890
C09900=1091.259,409.955,-100.076,178.161,25.082,153.892
C09901=1091.265,410.202,-100.116,178.165,25.091,153.893
C09902=1091.272,410.448,-100.156,178.168,25.099,153.895
C09903=1091.277,410.673,-100.193,178.171,25.107,153.897
C09904=1091.283,410.897,-100.230,178.173,25.115,153.898
C09905=1091.288,411.121,-100.267,178.176,25.123,153.900
C09906=1091.294,411.346,-100.303,178.179,25.131,153.902
C09907=1091.299,411.570,-100.340,178.182,25.139,153.903
C09908=1091.306,411.794,-100.377,178.184,25.147,153.905
C09909=1091.311,412.018,-100.414,178.188,25.156,153.907
C09910=1091.317,412.243,-100.450,178.191,25.164,153.908
C09911=1091.322,412.490,-100.491,178.193,25.172,153.910
C09912=1091.329,412.736,-100.532,178.197,25.182,153.912
C09913=1091.335,412.982,-100.572,178.200,25.191,153.914
C09914=1091.341,413.229,-100.613,178.203,25.199,153.915
C09915=1091.348,413.476,-100.653,178.206,25.209,153.917
C09916=1091.354,413.722,-100.695,178.209,25.218,153.919
C09917=1091.360,413.969,-100.735,178.213,25.227,153.921
C09918=1091.367,414.215,-100.775,178.215,25.236,153.923
C09919=1091.373,414.462,-100.816,178.219,25.245,153.925
C09920=1091.380,414.709,-100.857,178.222,25.254,153.927
C09921=1091.385,414.956,-100.898,178.225,25.264,153.928
C09922=1091.392,415.202,-100.939,178.228,25.272,153.930
C09923=1091.398,415.448,-100.979,178.231,25.282,153.932
C09924=1091.405,415.695,-101.021,178.235,25.291,153.934
C09925=1091.411,415.942,-101.061,178.238,25.301,153.936
C09926=1091.417,416.188,-101.102,178.241,25.310,153.938
C09927=1091.424,416.434,-101.142,178.244,25.319,153.940
C09928=1091.430,416.681,-101.184,178.247,25.329,153.942
C09929=1091.436,416.928,-101.225,178.250,25.339,153.944
C09930=1091.443,417.174,-101.266,178.254,25.348,153.946
C09931=1091.448,417.421,-101.306,178.257,25.357,153.948
C09932=1091.455,417.668,-101.348,178.260,25.367,153.950
C09933=1091.461,417.913,-101.389,178.264,25.377,153.952
C09934=1091.467,418.160,-101.430,178.266,25.386,153.954
C09935=1091.474,418.407,-101.472,178.269,25.396,153.956
C09936=1091.480,418.653,-101.513,178.273,25.405,153.958
C09937=1091.486,418.899,-101.554,178.276,25.416,153.960
C09938=1091.493,419.146,-101.596,178.279,25.425,153.962
C09939=1091.498,419.393,-101.637,178.283,25.435,153.964
C09940=1091.505,419.639,-101.677,178.286,25.445,153.966
C09941=1091.512,419.886,-101.719,178.289,25.455,153.968
C09942=1091.518,420.132,-101.761,178.292,25.465,153.970
C09943=1091.524,420.378,-101.802,178.296,25.474,153.972
C09944=1091.531,420.625,-101.843,178.299,25.485,153.974
C09945=1091.537,420.871,-101.885,178.302,25.495,153.976
C09946=1091.543,421.118,-101.927,178.305,25.504,153.978
C09947=1091.549,421.364,-101.968,178.308,25.514,153.980
C09948=1091.555,421.610,-102.010,178.311,25.524,153.982
C09949=1091.563,421.857,-102.051,178.314,25.534,153.984
C09950=1091.569,422.103,-102.092,178.317,25.544,153.987
C09951=1091.575,422.350,-102.134,178.321,25.554,153.989
C09952=1091.581,422.596,-102.176,178.325,25.565,153.991
C09953=1091.588,422.843,-102.217,178.328,25.575,153.993
C09954=1091.594,423.089,-102.260,178.331,25.586,153.995
C09955=1091.600,423.336,-102.301,178.334,25.596,153.997
C09956=1091.606,423.582,-102.343,178.338,25.606,154.000
C09957=1091.613,423.829,-102.385,178.341,25.617,154.002
C09958=1091.619,424.074,-102.427,178.344,25.627,154.004
C09959=1091.625,424.306,-102.466,178.347,25.637,154.006
C09960=1091.631,424.538,-102.505,178.350,25.647,154.008
C09961=1091.638,424.769,-102.545,178.353,25.657,154.010
C09962=1091.643,425.002,-102.584,178.356,25.667,154.012
C09963=1091.649,425.233,-102.624,178.358,25.676,154.015
C09964=1091.655,425.465,-102.663,178.362,25.686,154.017
C09965=1091.662,425.696,-102.703,178.365,25.697,154.019
C09966=1091.667,425.929,-102.743,178.368,25.707,154.021
C09967=1091.673,426.174,-102.785,178.371,25.717,154.023
C09968=1091.680,426.421,-102.827,178.375,25.728,154.025
C09969=1091.686,426.667,-102.869,178.378,25.739,154.028
C09970=1091.693,426.913,-102.911,178.381,25.750,154.030
C09971=1091.699,427.160,-102.953,178.385,25.760,154.032
C09972=1091.706,427.406,-102.996,178.388,25.771,154.035
C09973=1091.712,427.652,-103.038,178.391,25.782,154.037
C09974=1091.718,427.899,-103.080,178.394,25.793,154.039
C09975=1091.725,428.145,-103.123,178.397,25.804,154.042
C09976=1091.731,428.391,-103.165,178.401,25.815,154.044
C09977=1091.738,428.637,-103.207,178.404,25.826,154.046
C09978=1091.745,428.884,-103.249,178.407,25.837,154.049
C09979=1091.751,429.129,-103.291,178.410,25.848,154.051
C09980=1091.757,429.376,-103.335,178.414,25.860,154.054
C09981=1091.764,429.622,-103.377,178.417,25.871,154.056
C09982=1091.770,429.868,-103.419,178.420,25.882,154.059
C09983=1091.776,430.115,-103.462,178.423,25.893,154.061
C09984=1091.783,430.361,-103.505,178.428,25.905,154.063
C09985=1091.790,430.607,-103.548,178.431,25.916,154.066
C09986=1091.795,430.853,-103.590,178.433,25.928,154.068
C09987=1091.802,431.099,-103.633,178.437,25.939,154.071
C09988=1091.808,431.346,-103.676,178.440,25.951,154.073
C09989=1091.815,431.592,-103.718,178.443,25.962,154.076
C09990=1091.822,431.838,-103.761,178.446,25.973,154.078
C09991=1091.828,432.084,-103.805,178.450,25.985,154.081
C09992=1091.835,432.330,-103.847,178.453,25.997,154.083
C09993=1091.841,432.577,-103.890,178.457,26.009,154.086
C09994=1091.848,432.823,-103.933,178.460,26.021,154.089
C09995=1091.854,433.068,-103.976,178.463,26.032,154.091
C09996=1091.861,433.314,-104.019,178.467,26.044,154.094
//INST
///DATE 2021/06/17 10:54
///ATTR SC,RW,RJ
////FRAME ROBOT
///GROUP1 RB1
NOP
MOVL C00000 V=800.0 PL=0
MOVL C00001 V=800.0 PL=0
MOVL C00002 V=800.0 PL=0
MOVL C00003 V=800.0 PL=0
MOVL C00004 V=800.0 PL=0
MOVL C00005 V=800.0 PL=0
MOVL C00006 V=800.0 PL=0
MOVL C00007 V=800.0 PL=0
MOVL C00008 V=800.0 PL=0
MOVL C00009 V=800.0 PL=0
MOVL C00010 V=800.0 PL=0
MOVL C00011 V=800.0 PL=0
MOVL C00012 V=800.0 PL=0
MOVL C00013 V=800.0 PL=0
MOVL C00014 V=800.0 PL=0
MOVL C00015 V=800.0 PL=0
MOVL C00016 V=800.0 PL=0
MOVL C00017 V=800.0 PL=0
MOVL C00018 V=800.0 PL=0
MOVL C00019 V=800.0 PL=0
MOVL C00020 V=800.0 PL=0
MOVL C00021 V=800.0 PL=0
MOVL C00022 V=800.0 PL=0
MOVL C00023 V=800.0 PL=0
MOVL C00024 V=800.0 PL=0
MOVL C00025 V=800.0 PL=0
MOVL C00026 V=800.0 PL=0
MOVL C00027 V=800.0 PL=0
MOVL C00028 V=800.0 PL=0
MOVL C00029 V=800.0 PL=0
MOVL C00030 V=800.0 PL=0
MOVL C00031 V=800.0 PL=0
MOVL C00032 V=800.0 PL=0
MOVL C00033 V=800.0 PL=0
MOVL C00034 V=800.0 PL=0
MOVL C00035 V=800.0 PL=0
MOVL C00036 V=800.0 PL=0
MOVL C00037 V=800.0 PL=0
MOVL C00038 V=800.0 PL=0
MOVL C00039 V=800.0 PL=0
MOVL C00040 V=800.0 PL=0
MOVL C00041 V=800.0 PL=0
MOVL C00042 V=800.0 PL=0
MOVL C00043 V=800.0 PL=0
MOVL C00044 V=800.0 PL=0
MOVL C00045 V=800.0 PL=0
MOVL C00046 V=800.0 PL=0
MOVL C00047 V=800.0 PL=0
MOVL C00048 V=800.0 PL=0
MOVL C00049 V=800.0 PL=0
MOVL C00050 V=800.0 PL=0
MOVL C00051 V=800.0 PL=0
MOVL C00052 V=800.0 PL=0
MOVL C00053 V=800.0 PL=0
MOVL C00054 V=800.0 PL=0
MOVL C00055 V=800.0 PL=0
MOVL C00056 V=800.0 PL=0
MOVL C00057 V=800.0 PL=0
MOVL C00058 V=800.0 PL=0
MOVL C00059 V=800.0 PL=0
MOVL C00060 V=800.0 PL=0
MOVL C00061 V=800.0 PL=0
MOVL C00062 V=800.0 PL=0
MOVL C00063 V=800.0 PL=0
MOVL C00064 V=800.0 PL=0
MOVL C00065 V=800.0 PL=0
MOVL C00066 V=800.0 PL=0
MOVL C00067 V=800.0 PL=0
MOVL C00068 V=800.0 PL=0
MOVL C00069 V=800.0 PL=0
MOVL C00070 V=800.0 PL=0
MOVL C00071 V=800.0 PL=0
MOVL C00072 V=800.0 PL=0
MOVL C00073 V=800.0 PL=0
MOVL C00074 V=800.0 PL=0
MOVL C00075 V=800.0 PL=0
MOVL C00076 V=800.0 PL=0
MOVL C00077 V=800.0 PL=0
MOVL C00078 V=800.0 PL=0
MOVL C00079 V=800.0 PL=0
MOVL C00080 V=800.0 PL=0
MOVL C00081 V=800.0 PL=0
MOVL C00082 V=800.0 PL=0
MOVL C00083 V=800.0 PL=0
MOVL C00084 V=800.0 PL=0
MOVL C00085 V=800.0 PL=0
MOVL C00086 V=800.0 PL=0
MOVL C00087 V=800.0 PL=0
MOVL C00088 V=800.0 PL=0
MOVL C00089 V=800.0 PL=0
MOVL C00090 V=800.0 PL=0
MOVL C00091 V=800.0 PL=0
MOVL C00092 V=800.0 PL=0
MOVL C00093 V=800.0 PL=0
MOVL C00094 V=800.0 PL=0
MOVL C00095 V=800.0 PL=0
MOVL C00096 V=800.0 PL=0
MOVL C00097 V=800.0 PL=0
MOVL C00098 V=800.0 PL=0
MOVL C00099 V=800.0 PL=0
MOVL C00100 V=800.0 PL=0
MOVL C00101 V=800.0 PL=0
MOVL C00102 V=800.0 PL=0
MOVL C00103 V=800.0 PL=0
MOVL C00104 V=800.0 PL=0
MOVL C00105 V=800.0 PL=0
MOVL C00106 V=800.0 PL=0
MOVL C00107 V=800.0 PL=0
MOVL C00108 V=800.0 PL=0
MOVL C00109 V=800.0 PL=0
MOVL C00110 V=800.0 PL=0
MOVL C00111 V=800.0 PL=0
MOVL C00112 V=800.0 PL=0
MOVL C00113 V=800.0 PL=0
MOVL C00114 V=800.0 PL=0
MOVL C00115 V=800.0 PL=0
MOVL C00116 V=800.0 PL=0
MOVL C00117 V=800.0 PL=0
MOVL C00118 V=800.0 PL=0
MOVL C00119 V=800.0 PL=0
MOVL C00120 V=800.0 PL=0
MOVL C00121 V=800.0 PL=0
MOVL C00122 V=800.0 PL=0
MOVL C00123 V=800.0 PL=0
MOVL C00124 V=800.0 PL=0
MOVL C00125 V=800.0 PL=0
MOVL C00126 V=800.0 PL=0
MOVL C00127 V=800.0 PL=0
MOVL C00128 V=800.0 PL=0
MOVL C00129 V=800.0 PL=0
MOVL C00130 V=800.0 PL=0
MOVL C00131 V=800.0 PL=0
MOVL C00132 V=800.0 PL=0
MOVL C00133 V=800.0 PL=0
MOVL C00134 V=800.0 PL=0
MOVL C00135 V=800.0 PL=0
MOVL C00136 V=800.0 PL=0
MOVL C00137 V=800.0 PL=0
MOVL C00138 V=800.0 PL=0
MOVL C00139 V=800.0 PL=0
MOVL C00140 V=800.0 PL=0
MOVL C00141 V=800.0 PL=0
MOVL C00142 V=800.0 PL=0
MOVL C00143 V=800.0 PL=0
MOVL C00144 V=800.0 PL=0
MOVL C00145 V=800.0 PL=0
MOVL C00146 V=800.0 PL=0
MOVL C00147 V=800.0 PL=0
MOVL C00148 V=800.0 PL=0
MOVL C00149 V=800.0 PL=0
MOVL C00150 V=800.0 PL=0
MOVL C00151 V=800.0 PL=0
MOVL C00152 V=800.0 PL=0
MOVL C00153 V=800.0 PL=0
MOVL C00154 V=800.0 PL=0
MOVL C00155 V=800.0 PL=0
MOVL C00156 V=800.0 PL=0
MOVL C00157 V=800.0 PL=0
MOVL C00158 V=800.0 PL=0
MOVL C00159 V=800.0 PL=0
MOVL C00160 V=800.0 PL=0
MOVL C00161 V=800.0 PL=0
MOVL C00162 V=800.0 PL=0
MOVL C00163 V=800.0 PL=0
MOVL C00164 V=800.0 PL=0
MOVL C00165 V=800.0 PL=0
MOVL C00166 V=800.0 PL=0
MOVL C00167 V=800.0 PL=0
MOVL C00168 V=800.0 PL=0
MOVL C00169 V=800.0 PL=0
MOVL C00170 V=800.0 PL=0
MOVL C00171 V=800.0 PL=0
MOVL C00172 V=800.0 PL=0
MOVL C00173 V=800.0 PL=0
MOVL C00174 V=800.0 PL=0
MOVL C00175 V=800.0 PL=0
MOVL C00176 V=800.0 PL=0
MOVL C00177 V=800.0 PL=0
MOVL C00178 V=800.0 PL=0
MOVL C00179 V=800.0 PL=0
MOVL C00180 V=800.0 PL=0
MOVL C00181 V=800.0 PL=0
MOVL C00182 V=800.0 PL=0
MOVL C00183 V=800.0 PL=0
MOVL C00184 V=800.0 PL=0
MOVL C00185 V=800.0 PL=0
MOVL C00186 V=800.0 PL=0
MOVL C00187 V=800.0 PL=0
MOVL C00188 V=800.0 PL=0
MOVL C00189 V=800.0 PL=0
MOVL C00190 V=800.0 PL=0
MOVL C00191 V=800.0 PL=0
MOVL C00192 V=800.0 PL=0
MOVL C00193 V=800.0 PL=0
MOVL C00194 V=800.0 PL=0
MOVL C00195 V=800.0 PL=0
MOVL C00196 V=800.0 PL=0
MOVL C00197 V=800.0 PL=0
MOVL C00198 V=800.0 PL=0
MOVL C00199 V=800.0 PL=0
MOVL C00200 V=800.0 PL=0
MOVL C00201 V=800.0 PL=0
MOVL C00202 V=800.0 PL=0
MOVL C00203 V=800.0 PL=0
MOVL C00204 V=800.0 PL=0
MOVL C00205 V=800.0 PL=0
MOVL C00206 V=800.0 PL=0
MOVL C00207 V=800.0 PL=0
MOVL C00208 V=800.0 PL=0
MOVL C00209 V=800.0 PL=0
MOVL C00210 V=800.0 PL=0
MOVL C00211 V=800.0 PL=0
MOVL C00212 V=800.0 PL=0
MOVL C00213 V=800.0 PL=0
MOVL C00214 V=800.0 PL=0
MOVL C00215 V=800.0 PL=0
MOVL C00216 V=800.0 PL=0
MOVL C00217 V=800.0 PL=0
MOVL C00218 V=800.0 PL=0
MOVL C00219 V=800.0 PL=0
MOVL C00220 V=800.0 PL=0
MOVL C00221 V=800.0 PL=0
MOVL C00222 V=800.0 PL=0
MOVL C00223 V=800.0 PL=0
MOVL C00224 V=800.0 PL=0
MOVL C00225 V=800.0 PL=0
MOVL C00226 V=800.0 PL=0
MOVL C00227 V=800.0 PL=0
MOVL C00228 V=800.0 PL=0
MOVL C00229 V=800.0 PL=0
MOVL C00230 V=800.0 PL=0
MOVL C00231 V=800.0 PL=0
MOVL C00232 V=800.0 PL=0
MOVL C00233 V=800.0 PL=0
MOVL C00234 V=800.0 PL=0
MOVL C00235 V=800.0 PL=0
MOVL C00236 V=800.0 PL=0
MOVL C00237 V=800.0 PL=0
MOVL C00238 V=800.0 PL=0
MOVL C00239 V=800.0 PL=0
MOVL C00240 V=800.0 PL=0
MOVL C00241 V=800.0 PL=0
MOVL C00242 V=800.0 PL=0
MOVL C00243 V=800.0 PL=0
MOVL C00244 V=800.0 PL=0
MOVL C00245 V=800.0 PL=0
MOVL C00246 V=800.0 PL=0
MOVL C00247 V=800.0 PL=0
MOVL C00248 V=800.0 PL=0
MOVL C00249 V=800.0 PL=0
MOVL C00250 V=800.0 PL=0
MOVL C00251 V=800.0 PL=0
MOVL C00252 V=800.0 PL=0
MOVL C00253 V=800.0 PL=0
MOVL C00254 V=800.0 PL=0
MOVL C00255 V=800.0 PL=0
MOVL C00256 V=800.0 PL=0
MOVL C00257 V=800.0 PL=0
MOVL C00258 V=800.0 PL=0
MOVL C00259 V=800.0 PL=0
MOVL C00260 V=800.0 PL=0
MOVL C00261 V=800.0 PL=0
MOVL C00262 V=800.0 PL=0
MOVL C00263 V=800.0 PL=0
MOVL C00264 V=800.0 PL=0
MOVL C00265 V=800.0 PL=0
MOVL C00266 V=800.0 PL=0
MOVL C00267 V=800.0 PL=0
MOVL C00268 V=800.0 PL=0
MOVL C00269 V=800.0 PL=0
MOVL C00270 V=800.0 PL=0
MOVL C00271 V=800.0 PL=0
MOVL C00272 V=800.0 PL=0
MOVL C00273 V=800.0 PL=0
MOVL C00274 V=800.0 PL=0
MOVL C00275 V=800.0 PL=0
MOVL C00276 V=800.0 PL=0
MOVL C00277 V=800.0 PL=0
MOVL C00278 V=800.0 PL=0
MOVL C00279 V=800.0 PL=0
MOVL C00280 V=800.0 PL=0
MOVL C00281 V=800.0 PL=0
MOVL C00282 V=800.0 PL=0
MOVL C00283 V=800.0 PL=0
MOVL C00284 V=800.0 PL=0
MOVL C00285 V=800.0 PL=0
MOVL C00286 V=800.0 PL=0
MOVL C00287 V=800.0 PL=0
MOVL C00288 V=800.0 PL=0
MOVL C00289 V=800.0 PL=0
MOVL C00290 V=800.0 PL=0
MOVL C00291 V=800.0 PL=0
MOVL C00292 V=800.0 PL=0
MOVL C00293 V=800.0 PL=0
MOVL C00294 V=800.0 PL=0
MOVL C00295 V=800.0 PL=0
MOVL C00296 V=800.0 PL=0
MOVL C00297 V=800.0 PL=0
MOVL C00298 V=800.0 PL=0
MOVL C00299 V=800.0 PL=0
MOVL C00300 V=800.0 PL=0
MOVL C00301 V=800.0 PL=0
MOVL C00302 V=800.0 PL=0
MOVL C00303 V=800.0 PL=0
MOVL C00304 V=800.0 PL=0
MOVL C00305 V=800.0 PL=0
MOVL C00306 V=800.0 PL=0
MOVL C00307 V=800.0 PL=0
MOVL C00308 V=800.0 PL=0
MOVL C00309 V=800.0 PL=0
MOVL C00310 V=800.0 PL=0
MOVL C00311 V=800.0 PL=0
MOVL C00312 V=800.0 PL=0
MOVL C00313 V=800.0 PL=0
MOVL C00314 V=800.0 PL=0
MOVL C00315 V=800.0 PL=0
MOVL C00316 V=800.0 PL=0
MOVL C00317 V=800.0 PL=0
MOVL C00318 V=800.0 PL=0
MOVL C00319 V=800.0 PL=0
MOVL C00320 V=800.0 PL=0
MOVL C00321 V=800.0 PL=0
MOVL C00322 V=800.0 PL=0
MOVL C00323 V=800.0 PL=0
MOVL C00324 V=800.0 PL=0
MOVL C00325 V=800.0 PL=0
MOVL C00326 V=800.0 PL=0
MOVL C00327 V=800.0 PL=0
MOVL C00328 V=800.0 PL=0
MOVL C00329 V=800.0 PL=0
MOVL C00330 V=800.0 PL=0
MOVL C00331 V=800.0 PL=0
MOVL C00332 V=800.0 PL=0
MOVL C00333 V=800.0 PL=0
MOVL C00334 V=800.0 PL=0
MOVL C00335 V=800.0 PL=0
MOVL C00336 V=800.0 PL=0
MOVL C00337 V=800.0 PL=0
MOVL C00338 V=800.0 PL=0
MOVL C00339 V=800.0 PL=0
MOVL C00340 V=800.0 PL=0
MOVL C00341 V=800.0 PL=0
MOVL C00342 V=800.0 PL=0
MOVL C00343 V=800.0 PL=0
MOVL C00344 V=800.0 PL=0
MOVL C00345 V=800.0 PL=0
MOVL C00346 V=800.0 PL=0
MOVL C00347 V=800.0 PL=0
MOVL C00348 V=800.0 PL=0
MOVL C00349 V=800.0 PL=0
MOVL C00350 V=800.0 PL=0
MOVL C00351 V=800.0 PL=0
MOVL C00352 V=800.0 PL=0
MOVL C00353 V=800.0 PL=0
MOVL C00354 V=800.0 PL=0
MOVL C00355 V=800.0 PL=0
MOVL C00356 V=800.0 PL=0
MOVL C00357 V=800.0 PL=0
MOVL C00358 V=800.0 PL=0
MOVL C00359 V=800.0 PL=0
MOVL C00360 V=800.0 PL=0
MOVL C00361 V=800.0 PL=0
MOVL C00362 V=800.0 PL=0
MOVL C00363 V=800.0 PL=0
MOVL C00364 V=800.0 PL=0
MOVL C00365 V=800.0 PL=0
MOVL C00366 V=800.0 PL=0
MOVL C00367 V=800.0 PL=0
MOVL C00368 V=800.0 PL=0
MOVL C00369 V=800.0 PL=0
MOVL C00370 V=800.0 PL=0
MOVL C00371 V=800.0 PL=0
MOVL C00372 V=800.0 PL=0
MOVL C00373 V=800.0 PL=0
MOVL C00374 V=800.0 PL=0
MOVL C00375 V=800.0 PL=0
MOVL C00376 V=800.0 PL=0
MOVL C00377 V=800.0 PL=0
MOVL C00378 V=800.0 PL=0
MOVL C00379 V=800.0 PL=0
MOVL C00380 V=800.0 PL=0
MOVL C00381 V=800.0 PL=0
MOVL C00382 V=800.0 PL=0
MOVL C00383 V=800.0 PL=0
MOVL C00384 V=800.0 PL=0
MOVL C00385 V=800.0 PL=0
MOVL C00386 V=800.0 PL=0
MOVL C00387 V=800.0 PL=0
MOVL C00388 V=800.0 PL=0
MOVL C00389 V=800.0 PL=0
MOVL C00390 V=800.0 PL=0
MOVL C00391 V=800.0 PL=0
MOVL C00392 V=800.0 PL=0
MOVL C00393 V=800.0 PL=0
MOVL C00394 V=800.0 PL=0
MOVL C00395 V=800.0 PL=0
MOVL C00396 V=800.0 PL=0
MOVL C00397 V=800.0 PL=0
MOVL C00398 V=800.0 PL=0
MOVL C00399 V=800.0 PL=0
MOVL C00400 V=800.0 PL=0
MOVL C00401 V=800.0 PL=0
MOVL C00402 V=800.0 PL=0
MOVL C00403 V=800.0 PL=0
MOVL C00404 V=800.0 PL=0
MOVL C00405 V=800.0 PL=0
MOVL C00406 V=800.0 PL=0
MOVL C00407 V=800.0 PL=0
MOVL C00408 V=800.0 PL=0
MOVL C00409 V=800.0 PL=0
MOVL C00410 V=800.0 PL=0
MOVL C00411 V=800.0 PL=0
MOVL C00412 V=800.0 PL=0
MOVL C00413 V=800.0 PL=0
MOVL C00414 V=800.0 PL=0
MOVL C00415 V=800.0 PL=0
MOVL C00416 V=800.0 PL=0
MOVL C00417 V=800.0 PL=0
MOVL C00418 V=800.0 PL=0
MOVL C00419 V=800.0 PL=0
MOVL C00420 V=800.0 PL=0
MOVL C00421 V=800.0 PL=0
MOVL C00422 V=800.0 PL=0
MOVL C00423 V=800.0 PL=0
MOVL C00424 V=800.0 PL=0
MOVL C00425 V=800.0 PL=0
MOVL C00426 V=800.0 PL=0
MOVL C00427 V=800.0 PL=0
MOVL C00428 V=800.0 PL=0
MOVL C00429 V=800.0 PL=0
MOVL C00430 V=800.0 PL=0
MOVL C00431 V=800.0 PL=0
MOVL C00432 V=800.0 PL=0
MOVL C00433 V=800.0 PL=0
MOVL C00434 V=800.0 PL=0
MOVL C00435 V=800.0 PL=0
MOVL C00436 V=800.0 PL=0
MOVL C00437 V=800.0 PL=0
MOVL C00438 V=800.0 PL=0
MOVL C00439 V=800.0 PL=0
MOVL C00440 V=800.0 PL=0
MOVL C00441 V=800.0 PL=0
MOVL C00442 V=800.0 PL=0
MOVL C00443 V=800.0 PL=0
MOVL C00444 V=800.0 PL=0
MOVL C00445 V=800.0 PL=0
MOVL C00446 V=800.0 PL=0
MOVL C00447 V=800.0 PL=0
MOVL C00448 V=800.0 PL=0
MOVL C00449 V=800.0 PL=0
MOVL C00450 V=800.0 PL=0
MOVL C00451 V=800.0 PL=0
MOVL C00452 V=800.0 PL=0
MOVL C00453 V=800.0 PL=0
MOVL C00454 V=800.0 PL=0
MOVL C00455 V=800.0 PL=0
MOVL C00456 V=800.0 PL=0
MOVL C00457 V=800.0 PL=0
MOVL C00458 V=800.0 PL=0
MOVL C00459 V=800.0 PL=0
MOVL C00460 V=800.0 PL=0
MOVL C00461 V=800.0 PL=0
MOVL C00462 V=800.0 PL=0
MOVL C00463 V=800.0 PL=0
MOVL C00464 V=800.0 PL=0
MOVL C00465 V=800.0 PL=0
MOVL C00466 V=800.0 PL=0
MOVL C00467 V=800.0 PL=0
MOVL C00468 V=800.0 PL=0
MOVL C00469 V=800.0 PL=0
MOVL C00470 V=800.0 PL=0
MOVL C00471 V=800.0 PL=0
MOVL C00472 V=800.0 PL=0
MOVL C00473 V=800.0 PL=0
MOVL C00474 V=800.0 PL=0
MOVL C00475 V=800.0 PL=0
MOVL C00476 V=800.0 PL=0
MOVL C00477 V=800.0 PL=0
MOVL C00478 V=800.0 PL=0
MOVL C00479 V=800.0 PL=0
MOVL C00480 V=800.0 PL=0
MOVL C00481 V=800.0 PL=0
MOVL C00482 V=800.0 PL=0
MOVL C00483 V=800.0 PL=0
MOVL C00484 V=800.0 PL=0
MOVL C00485 V=800.0 PL=0
MOVL C00486 V=800.0 PL=0
MOVL C00487 V=800.0 PL=0
MOVL C00488 V=800.0 PL=0
MOVL C00489 V=800.0 PL=0
MOVL C00490 V=800.0 PL=0
MOVL C00491 V=800.0 PL=0
MOVL C00492 V=800.0 PL=0
MOVL C00493 V=800.0 PL=0
MOVL C00494 V=800.0 PL=0
MOVL C00495 V=800.0 PL=0
MOVL C00496 V=800.0 PL=0
MOVL C00497 V=800.0 PL=0
MOVL C00498 V=800.0 PL=0
MOVL C00499 V=800.0 PL=0
MOVL C00500 V=800.0 PL=0
MOVL C00501 V=800.0 PL=0
MOVL C00502 V=800.0 PL=0
MOVL C00503 V=800.0 PL=0
MOVL C00504 V=800.0 PL=0
MOVL C00505 V=800.0 PL=0
MOVL C00506 V=800.0 PL=0
MOVL C00507 V=800.0 PL=0
MOVL C00508 V=800.0 PL=0
MOVL C00509 V=800.0 PL=0
MOVL C00510 V=800.0 PL=0
MOVL C00511 V=800.0 PL=0
MOVL C00512 V=800.0 PL=0
MOVL C00513 V=800.0 PL=0
MOVL C00514 V=800.0 PL=0
MOVL C00515 V=800.0 PL=0
MOVL C00516 V=800.0 PL=0
MOVL C00517 V=800.0 PL=0
MOVL C00518 V=800.0 PL=0
MOVL C00519 V=800.0 PL=0
MOVL C00520 V=800.0 PL=0
MOVL C00521 V=800.0 PL=0
MOVL C00522 V=800.0 PL=0
MOVL C00523 V=800.0 PL=0
MOVL C00524 V=800.0 PL=0
MOVL C00525 V=800.0 PL=0
MOVL C00526 V=800.0 PL=0
MOVL C00527 V=800.0 PL=0
MOVL C00528 V=800.0 PL=0
MOVL C00529 V=800.0 PL=0
MOVL C00530 V=800.0 PL=0
MOVL C00531 V=800.0 PL=0
MOVL C00532 V=800.0 PL=0
MOVL C00533 V=800.0 PL=0
MOVL C00534 V=800.0 PL=0
MOVL C00535 V=800.0 PL=0
MOVL C00536 V=800.0 PL=0
MOVL C00537 V=800.0 PL=0
MOVL C00538 V=800.0 PL=0
MOVL C00539 V=800.0 PL=0
MOVL C00540 V=800.0 PL=0
MOVL C00541 V=800.0 PL=0
MOVL C00542 V=800.0 PL=0
MOVL C00543 V=800.0 PL=0
MOVL C00544 V=800.0 PL=0
MOVL C00545 V=800.0 PL=0
MOVL C00546 V=800.0 PL=0
MOVL C00547 V=800.0 PL=0
MOVL C00548 V=800.0 PL=0
MOVL C00549 V=800.0 PL=0
MOVL C00550 V=800.0 PL=0
MOVL C00551 V=800.0 PL=0
MOVL C00552 V=800.0 PL=0
MOVL C00553 V=800.0 PL=0
MOVL C00554 V=800.0 PL=0
MOVL C00555 V=800.0 PL=0
MOVL C00556 V=800.0 PL=0
MOVL C00557 V=800.0 PL=0
MOVL C00558 V=800.0 PL=0
MOVL C00559 V=800.0 PL=0
MOVL C00560 V=800.0 PL=0
MOVL C00561 V=800.0 PL=0
MOVL C00562 V=800.0 PL=0
MOVL C00563 V=800.0 PL=0
MOVL C00564 V=800.0 PL=0
MOVL C00565 V=800.0 PL=0
MOVL C00566 V=800.0 PL=0
MOVL C00567 V=800.0 PL=0
MOVL C00568 V=800.0 PL=0
MOVL C00569 V=800.0 PL=0
MOVL C00570 V=800.0 PL=0
MOVL C00571 V=800.0 PL=0
MOVL C00572 V=800.0 PL=0
MOVL C00573 V=800.0 PL=0
MOVL C00574 V=800.0 PL=0
MOVL C00575 V=800.0 PL=0
MOVL C00576 V=800.0 PL=0
MOVL C00577 V=800.0 PL=0
MOVL C00578 V=800.0 PL=0
MOVL C00579 V=800.0 PL=0
MOVL C00580 V=800.0 PL=0
MOVL C00581 V=800.0 PL=0
MOVL C00582 V=800.0 PL=0
MOVL C00583 V=800.0 PL=0
MOVL C00584 V=800.0 PL=0
MOVL C00585 V=800.0 PL=0
MOVL C00586 V=800.0 PL=0
MOVL C00587 V=800.0 PL=0
MOVL C00588 V=800.0 PL=0
MOVL C00589 V=800.0 PL=0
MOVL C00590 V=800.0 PL=0
MOVL C00591 V=800.0 PL=0
MOVL C00592 V=800.0 PL=0
MOVL C00593 V=800.0 PL=0
MOVL C00594 V=800.0 PL=0
MOVL C00595 V=800.0 PL=0
MOVL C00596 V=800.0 PL=0
MOVL C00597 V=800.0 PL=0
MOVL C00598 V=800.0 PL=0
MOVL C00599 V=800.0 PL=0
MOVL C00600 V=800.0 PL=0
MOVL C00601 V=800.0 PL=0
MOVL C00602 V=800.0 PL=0
MOVL C00603 V=800.0 PL=0
MOVL C00604 V=800.0 PL=0
MOVL C00605 V=800.0 PL=0
MOVL C00606 V=800.0 PL=0
MOVL C00607 V=800.0 PL=0
MOVL C00608 V=800.0 PL=0
MOVL C00609 V=800.0 PL=0
MOVL C00610 V=800.0 PL=0
MOVL C00611 V=800.0 PL=0
MOVL C00612 V=800.0 PL=0
MOVL C00613 V=800.0 PL=0
MOVL C00614 V=800.0 PL=0
MOVL C00615 V=800.0 PL=0
MOVL C00616 V=800.0 PL=0
MOVL C00617 V=800.0 PL=0
MOVL C00618 V=800.0 PL=0
MOVL C00619 V=800.0 PL=0
MOVL C00620 V=800.0 PL=0
MOVL C00621 V=800.0 PL=0
MOVL C00622 V=800.0 PL=0
MOVL C00623 V=800.0 PL=0
MOVL C00624 V=800.0 PL=0
MOVL C00625 V=800.0 PL=0
MOVL C00626 V=800.0 PL=0
MOVL C00627 V=800.0 PL=0
MOVL C00628 V=800.0 PL=0
MOVL C00629 V=800.0 PL=0
MOVL C00630 V=800.0 PL=0
MOVL C00631 V=800.0 PL=0
MOVL C00632 V=800.0 PL=0
MOVL C00633 V=800.0 PL=0
MOVL C00634 V=800.0 PL=0
MOVL C00635 V=800.0 PL=0
MOVL C00636 V=800.0 PL=0
MOVL C00637 V=800.0 PL=0
MOVL C00638 V=800.0 PL=0
MOVL C00639 V=800.0 PL=0
MOVL C00640 V=800.0 PL=0
MOVL C00641 V=800.0 PL=0
MOVL C00642 V=800.0 PL=0
MOVL C00643 V=800.0 PL=0
MOVL C00644 V=800.0 PL=0
MOVL C00645 V=800.0 PL=0
MOVL C00646 V=800.0 PL=0
MOVL C00647 V=800.0 PL=0
MOVL C00648 V=800.0 PL=0
MOVL C00649 V=800.0 PL=0
MOVL C00650 V=800.0 PL=0
MOVL C00651 V=800.0 PL=0
MOVL C00652 V=800.0 PL=0
MOVL C00653 V=800.0 PL=0
MOVL C00654 V=800.0 PL=0
MOVL C00655 V=800.0 PL=0
MOVL C00656 V=800.0 PL=0
MOVL C00657 V=800.0 PL=0
MOVL C00658 V=800.0 PL=0
MOVL C00659 V=800.0 PL=0
MOVL C00660 V=800.0 PL=0
MOVL C00661 V=800.0 PL=0
MOVL C00662 V=800.0 PL=0
MOVL C00663 V=800.0 PL=0
MOVL C00664 V=800.0 PL=0
MOVL C00665 V=800.0 PL=0
MOVL C00666 V=800.0 PL=0
MOVL C00667 V=800.0 PL=0
MOVL C00668 V=800.0 PL=0
MOVL C00669 V=800.0 PL=0
MOVL C00670 V=800.0 PL=0
MOVL C00671 V=800.0 PL=0
MOVL C00672 V=800.0 PL=0
MOVL C00673 V=800.0 PL=0
MOVL C00674 V=800.0 PL=0
MOVL C00675 V=800.0 PL=0
MOVL C00676 V=800.0 PL=0
MOVL C00677 V=800.0 PL=0
MOVL C00678 V=800.0 PL=0
MOVL C00679 V=800.0 PL=0
MOVL C00680 V=800.0 PL=0
MOVL C00681 V=800.0 PL=0
MOVL C00682 V=800.0 PL=0
MOVL C00683 V=800.0 PL=0
MOVL C00684 V=800.0 PL=0
MOVL C00685 V=800.0 PL=0
MOVL C00686 V=800.0 PL=0
MOVL C00687 V=800.0 PL=0
MOVL C00688 V=800.0 PL=0
MOVL C00689 V=800.0 PL=0
MOVL C00690 V=800.0 PL=0
MOVL C00691 V=800.0 PL=0
MOVL C00692 V=800.0 PL=0
MOVL C00693 V=800.0 PL=0
MOVL C00694 V=800.0 PL=0
MOVL C00695 V=800.0 PL=0
MOVL C00696 V=800.0 PL=0
MOVL C00697 V=800.0 PL=0
MOVL C00698 V=800.0 PL=0
MOVL C00699 V=800.0 PL=0
MOVL C00700 V=800.0 PL=0
MOVL C00701 V=800.0 PL=0
MOVL C00702 V=800.0 PL=0
MOVL C00703 V=800.0 PL=0
MOVL C00704 V=800.0 PL=0
MOVL C00705 V=800.0 PL=0
MOVL C00706 V=800.0 PL=0
MOVL C00707 V=800.0 PL=0
MOVL C00708 V=800.0 PL=0
MOVL C00709 V=800.0 PL=0
MOVL C00710 V=800.0 PL=0
MOVL C00711 V=800.0 PL=0
MOVL C00712 V=800.0 PL=0
MOVL C00713 V=800.0 PL=0
MOVL C00714 V=800.0 PL=0
MOVL C00715 V=800.0 PL=0
MOVL C00716 V=800.0 PL=0
MOVL C00717 V=800.0 PL=0
MOVL C00718 V=800.0 PL=0
MOVL C00719 V=800.0 PL=0
MOVL C00720 V=800.0 PL=0
MOVL C00721 V=800.0 PL=0
MOVL C00722 V=800.0 PL=0
MOVL C00723 V=800.0 PL=0
MOVL C00724 V=800.0 PL=0
MOVL C00725 V=800.0 PL=0
MOVL C00726 V=800.0 PL=0
MOVL C00727 V=800.0 PL=0
MOVL C00728 V=800.0 PL=0
MOVL C00729 V=800.0 PL=0
MOVL C00730 V=800.0 PL=0
MOVL C00731 V=800.0 PL=0
MOVL C00732 V=800.0 PL=0
MOVL C00733 V=800.0 PL=0
MOVL C00734 V=800.0 PL=0
MOVL C00735 V=800.0 PL=0
MOVL C00736 V=800.0 PL=0
MOVL C00737 V=800.0 PL=0
MOVL C00738 V=800.0 PL=0
MOVL C00739 V=800.0 PL=0
MOVL C00740 V=800.0 PL=0
MOVL C00741 V=800.0 PL=0
MOVL C00742 V=800.0 PL=0
MOVL C00743 V=800.0 PL=0
MOVL C00744 V=800.0 PL=0
MOVL C00745 V=800.0 PL=0
MOVL C00746 V=800.0 PL=0
MOVL C00747 V=800.0 PL=0
MOVL C00748 V=800.0 PL=0
MOVL C00749 V=800.0 PL=0
MOVL C00750 V=800.0 PL=0
MOVL C00751 V=800.0 PL=0
MOVL C00752 V=800.0 PL=0
MOVL C00753 V=800.0 PL=0
MOVL C00754 V=800.0 PL=0
MOVL C00755 V=800.0 PL=0
MOVL C00756 V=800.0 PL=0
MOVL C00757 V=800.0 PL=0
MOVL C00758 V=800.0 PL=0
MOVL C00759 V=800.0 PL=0
MOVL C00760 V=800.0 PL=0
MOVL C00761 V=800.0 PL=0
MOVL C00762 V=800.0 PL=0
MOVL C00763 V=800.0 PL=0
MOVL C00764 V=800.0 PL=0
MOVL C00765 V=800.0 PL=0
MOVL C00766 V=800.0 PL=0
MOVL C00767 V=800.0 PL=0
MOVL C00768 V=800.0 PL=0
MOVL C00769 V=800.0 PL=0
MOVL C00770 V=800.0 PL=0
MOVL C00771 V=800.0 PL=0
MOVL C00772 V=800.0 PL=0
MOVL C00773 V=800.0 PL=0
MOVL C00774 V=800.0 PL=0
MOVL C00775 V=800.0 PL=0
MOVL C00776 V=800.0 PL=0
MOVL C00777 V=800.0 PL=0
MOVL C00778 V=800.0 PL=0
MOVL C00779 V=800.0 PL=0
MOVL C00780 V=800.0 PL=0
MOVL C00781 V=800.0 PL=0
MOVL C00782 V=800.0 PL=0
MOVL C00783 V=800.0 PL=0
MOVL C00784 V=800.0 PL=0
MOVL C00785 V=800.0 PL=0
MOVL C00786 V=800.0 PL=0
MOVL C00787 V=800.0 PL=0
MOVL C00788 V=800.0 PL=0
MOVL C00789 V=800.0 PL=0
MOVL C00790 V=800.0 PL=0
MOVL C00791 V=800.0 PL=0
MOVL C00792 V=800.0 PL=0
MOVL C00793 V=800.0 PL=0
MOVL C00794 V=800.0 PL=0
MOVL C00795 V=800.0 PL=0
MOVL C00796 V=800.0 PL=0
MOVL C00797 V=800.0 PL=0
MOVL C00798 V=800.0 PL=0
MOVL C00799 V=800.0 PL=0
MOVL C00800 V=800.0 PL=0
MOVL C00801 V=800.0 PL=0
MOVL C00802 V=800.0 PL=0
MOVL C00803 V=800.0 PL=0
MOVL C00804 V=800.0 PL=0
MOVL C00805 V=800.0 PL=0
MOVL C00806 V=800.0 PL=0
MOVL C00807 V=800.0 PL=0
MOVL C00808 V=800.0 PL=0
MOVL C00809 V=800.0 PL=0
MOVL C00810 V=800.0 PL=0
MOVL C00811 V=800.0 PL=0
MOVL C00812 V=800.0 PL=0
MOVL C00813 V=800.0 PL=0
MOVL C00814 V=800.0 PL=0
MOVL C00815 V=800.0 PL=0
MOVL C00816 V=800.0 PL=0
MOVL C00817 V=800.0 PL=0
MOVL C00818 V=800.0 PL=0
MOVL C00819 V=800.0 PL=0
MOVL C00820 V=800.0 PL=0
MOVL C00821 V=800.0 PL=0
MOVL C00822 V=800.0 PL=0
MOVL C00823 V=800.0 PL=0
MOVL C00824 V=800.0 PL=0
MOVL C00825 V=800.0 PL=0
MOVL C00826 V=800.0 PL=0
MOVL C00827 V=800.0 PL=0
MOVL C00828 V=800.0 PL=0
MOVL C00829 V=800.0 PL=0
MOVL C00830 V=800.0 PL=0
MOVL C00831 V=800.0 PL=0
MOVL C00832 V=800.0 PL=0
MOVL C00833 V=800.0 PL=0
MOVL C00834 V=800.0 PL=0
MOVL C00835 V=800.0 PL=0
MOVL C00836 V=800.0 PL=0
MOVL C00837 V=800.0 PL=0
MOVL C00838 V=800.0 PL=0
MOVL C00839 V=800.0 PL=0
MOVL C00840 V=800.0 PL=0
MOVL C00841 V=800.0 PL=0
MOVL C00842 V=800.0 PL=0
MOVL C00843 V=800.0 PL=0
MOVL C00844 V=800.0 PL=0
MOVL C00845 V=800.0 PL=0
MOVL C00846 V=800.0 PL=0
MOVL C00847 V=800.0 PL=0
MOVL C00848 V=800.0 PL=0
MOVL C00849 V=800.0 PL=0
MOVL C00850 V=800.0 PL=0
MOVL C00851 V=800.0 PL=0
MOVL C00852 V=800.0 PL=0
MOVL C00853 V=800.0 PL=0
MOVL C00854 V=800.0 PL=0
MOVL C00855 V=800.0 PL=0
MOVL C00856 V=800.0 PL=0
MOVL C00857 V=800.0 PL=0
MOVL C00858 V=800.0 PL=0
MOVL C00859 V=800.0 PL=0
MOVL C00860 V=800.0 PL=0
MOVL C00861 V=800.0 PL=0
MOVL C00862 V=800.0 PL=0
MOVL C00863 V=800.0 PL=0
MOVL C00864 V=800.0 PL=0
MOVL C00865 V=800.0 PL=0
MOVL C00866 V=800.0 PL=0
MOVL C00867 V=800.0 PL=0
MOVL C00868 V=800.0 PL=0
MOVL C00869 V=800.0 PL=0
MOVL C00870 V=800.0 PL=0
MOVL C00871 V=800.0 PL=0
MOVL C00872 V=800.0 PL=0
MOVL C00873 V=800.0 PL=0
MOVL C00874 V=800.0 PL=0
MOVL C00875 V=800.0 PL=0
MOVL C00876 V=800.0 PL=0
MOVL C00877 V=800.0 PL=0
MOVL C00878 V=800.0 PL=0
MOVL C00879 V=800.0 PL=0
MOVL C00880 V=800.0 PL=0
MOVL C00881 V=800.0 PL=0
MOVL C00882 V=800.0 PL=0
MOVL C00883 V=800.0 PL=0
MOVL C00884 V=800.0 PL=0
MOVL C00885 V=800.0 PL=0
MOVL C00886 V=800.0 PL=0
MOVL C00887 V=800.0 PL=0
MOVL C00888 V=800.0 PL=0
MOVL C00889 V=800.0 PL=0
MOVL C00890 V=800.0 PL=0
MOVL C00891 V=800.0 PL=0
MOVL C00892 V=800.0 PL=0
MOVL C00893 V=800.0 PL=0
MOVL C00894 V=800.0 PL=0
MOVL C00895 V=800.0 PL=0
MOVL C00896 V=800.0 PL=0
MOVL C00897 V=800.0 PL=0
MOVL C00898 V=800.0 PL=0
MOVL C00899 V=800.0 PL=0
MOVL C00900 V=800.0 PL=0
MOVL C00901 V=800.0 PL=0
MOVL C00902 V=800.0 PL=0
MOVL C00903 V=800.0 PL=0
MOVL C00904 V=800.0 PL=0
MOVL C00905 V=800.0 PL=0
MOVL C00906 V=800.0 PL=0
MOVL C00907 V=800.0 PL=0
MOVL C00908 V=800.0 PL=0
MOVL C00909 V=800.0 PL=0
MOVL C00910 V=800.0 PL=0
MOVL C00911 V=800.0 PL=0
MOVL C00912 V=800.0 PL=0
MOVL C00913 V=800.0 PL=0
MOVL C00914 V=800.0 PL=0
MOVL C00915 V=800.0 PL=0
MOVL C00916 V=800.0 PL=0
MOVL C00917 V=800.0 PL=0
MOVL C00918 V=800.0 PL=0
MOVL C00919 V=800.0 PL=0
MOVL C00920 V=800.0 PL=0
MOVL C00921 V=800.0 PL=0
MOVL C00922 V=800.0 PL=0
MOVL C00923 V=800.0 PL=0
MOVL C00924 V=800.0 PL=0
MOVL C00925 V=800.0 PL=0
MOVL C00926 V=800.0 PL=0
MOVL C00927 V=800.0 PL=0
MOVL C00928 V=800.0 PL=0
MOVL C00929 V=800.0 PL=0
MOVL C00930 V=800.0 PL=0
MOVL C00931 V=800.0 PL=0
MOVL C00932 V=800.0 PL=0
MOVL C00933 V=800.0 PL=0
MOVL C00934 V=800.0 PL=0
MOVL C00935 V=800.0 PL=0
MOVL C00936 V=800.0 PL=0
MOVL C00937 V=800.0 PL=0
MOVL C00938 V=800.0 PL=0
MOVL C00939 V=800.0 PL=0
MOVL C00940 V=800.0 PL=0
MOVL C00941 V=800.0 PL=0
MOVL C00942 V=800.0 PL=0
MOVL C00943 V=800.0 PL=0
MOVL C00944 V=800.0 PL=0
MOVL C00945 V=800.0 PL=0
MOVL C00946 V=800.0 PL=0
MOVL C00947 V=800.0 PL=0
MOVL C00948 V=800.0 PL=0
MOVL C00949 V=800.0 PL=0
MOVL C00950 V=800.0 PL=0
MOVL C00951 V=800.0 PL=0
MOVL C00952 V=800.0 PL=0
MOVL C00953 V=800.0 PL=0
MOVL C00954 V=800.0 PL=0
MOVL C00955 V=800.0 PL=0
MOVL C00956 V=800.0 PL=0
MOVL C00957 V=800.0 PL=0
MOVL C00958 V=800.0 PL=0
MOVL C00959 V=800.0 PL=0
MOVL C00960 V=800.0 PL=0
MOVL C00961 V=800.0 PL=0
MOVL C00962 V=800.0 PL=0
MOVL C00963 V=800.0 PL=0
MOVL C00964 V=800.0 PL=0
MOVL C00965 V=800.0 PL=0
MOVL C00966 V=800.0 PL=0
MOVL C00967 V=800.0 PL=0
MOVL C00968 V=800.0 PL=0
MOVL C00969 V=800.0 PL=0
MOVL C00970 V=800.0 PL=0
MOVL C00971 V=800.0 PL=0
MOVL C00972 V=800.0 PL=0
MOVL C00973 V=800.0 PL=0
MOVL C00974 V=800.0 PL=0
MOVL C00975 V=800.0 PL=0
MOVL C00976 V=800.0 PL=0
MOVL C00977 V=800.0 PL=0
MOVL C00978 V=800.0 PL=0
MOVL C00979 V=800.0 PL=0
MOVL C00980 V=800.0 PL=0
MOVL C00981 V=800.0 PL=0
MOVL C00982 V=800.0 PL=0
MOVL C00983 V=800.0 PL=0
MOVL C00984 V=800.0 PL=0
MOVL C00985 V=800.0 PL=0
MOVL C00986 V=800.0 PL=0
MOVL C00987 V=800.0 PL=0
MOVL C00988 V=800.0 PL=0
MOVL C00989 V=800.0 PL=0
MOVL C00990 V=800.0 PL=0
MOVL C00991 V=800.0 PL=0
MOVL C00992 V=800.0 PL=0
MOVL C00993 V=800.0 PL=0
MOVL C00994 V=800.0 PL=0
MOVL C00995 V=800.0 PL=0
MOVL C00996 V=800.0 PL=0
MOVL C00997 V=800.0 PL=0
MOVL C00998 V=800.0 PL=0
MOVL C00999 V=800.0 PL=0
MOVL C01000 V=800.0 PL=0
MOVL C01001 V=800.0 PL=0
MOVL C01002 V=800.0 PL=0
MOVL C01003 V=800.0 PL=0
MOVL C01004 V=800.0 PL=0
MOVL C01005 V=800.0 PL=0
MOVL C01006 V=800.0 PL=0
MOVL C01007 V=800.0 PL=0
MOVL C01008 V=800.0 PL=0
MOVL C01009 V=800.0 PL=0
MOVL C01010 V=800.0 PL=0
MOVL C01011 V=800.0 PL=0
MOVL C01012 V=800.0 PL=0
MOVL C01013 V=800.0 PL=0
MOVL C01014 V=800.0 PL=0
MOVL C01015 V=800.0 PL=0
MOVL C01016 V=800.0 PL=0
MOVL C01017 V=800.0 PL=0
MOVL C01018 V=800.0 PL=0
MOVL C01019 V=800.0 PL=0
MOVL C01020 V=800.0 PL=0
MOVL C01021 V=800.0 PL=0
MOVL C01022 V=800.0 PL=0
MOVL C01023 V=800.0 PL=0
MOVL C01024 V=800.0 PL=0
MOVL C01025 V=800.0 PL=0
MOVL C01026 V=800.0 PL=0
MOVL C01027 V=800.0 PL=0
MOVL C01028 V=800.0 PL=0
MOVL C01029 V=800.0 PL=0
MOVL C01030 V=800.0 PL=0
MOVL C01031 V=800.0 PL=0
MOVL C01032 V=800.0 PL=0
MOVL C01033 V=800.0 PL=0
MOVL C01034 V=800.0 PL=0
MOVL C01035 V=800.0 PL=0
MOVL C01036 V=800.0 PL=0
MOVL C01037 V=800.0 PL=0
MOVL C01038 V=800.0 PL=0
MOVL C01039 V=800.0 PL=0
MOVL C01040 V=800.0 PL=0
MOVL C01041 V=800.0 PL=0
MOVL C01042 V=800.0 PL=0
MOVL C01043 V=800.0 PL=0
MOVL C01044 V=800.0 PL=0
MOVL C01045 V=800.0 PL=0
MOVL C01046 V=800.0 PL=0
MOVL C01047 V=800.0 PL=0
MOVL C01048 V=800.0 PL=0
MOVL C01049 V=800.0 PL=0
MOVL C01050 V=800.0 PL=0
MOVL C01051 V=800.0 PL=0
MOVL C01052 V=800.0 PL=0
MOVL C01053 V=800.0 PL=0
MOVL C01054 V=800.0 PL=0
MOVL C01055 V=800.0 PL=0
MOVL C01056 V=800.0 PL=0
MOVL C01057 V=800.0 PL=0
MOVL C01058 V=800.0 PL=0
MOVL C01059 V=800.0 PL=0
MOVL C01060 V=800.0 PL=0
MOVL C01061 V=800.0 PL=0
MOVL C01062 V=800.0 PL=0
MOVL C01063 V=800.0 PL=0
MOVL C01064 V=800.0 PL=0
MOVL C01065 V=800.0 PL=0
MOVL C01066 V=800.0 PL=0
MOVL C01067 V=800.0 PL=0
MOVL C01068 V=800.0 PL=0
MOVL C01069 V=800.0 PL=0
MOVL C01070 V=800.0 PL=0
MOVL C01071 V=800.0 PL=0
MOVL C01072 V=800.0 PL=0
MOVL C01073 V=800.0 PL=0
MOVL C01074 V=800.0 PL=0
MOVL C01075 V=800.0 PL=0
MOVL C01076 V=800.0 PL=0
MOVL C01077 V=800.0 PL=0
MOVL C01078 V=800.0 PL=0
MOVL C01079 V=800.0 PL=0
MOVL C01080 V=800.0 PL=0
MOVL C01081 V=800.0 PL=0
MOVL C01082 V=800.0 PL=0
MOVL C01083 V=800.0 PL=0
MOVL C01084 V=800.0 PL=0
MOVL C01085 V=800.0 PL=0
MOVL C01086 V=800.0 PL=0
MOVL C01087 V=800.0 PL=0
MOVL C01088 V=800.0 PL=0
MOVL C01089 V=800.0 PL=0
MOVL C01090 V=800.0 PL=0
MOVL C01091 V=800.0 PL=0
MOVL C01092 V=800.0 PL=0
MOVL C01093 V=800.0 PL=0
MOVL C01094 V=800.0 PL=0
MOVL C01095 V=800.0 PL=0
MOVL C01096 V=800.0 PL=0
MOVL C01097 V=800.0 PL=0
MOVL C01098 V=800.0 PL=0
MOVL C01099 V=800.0 PL=0
MOVL C01100 V=800.0 PL=0
MOVL C01101 V=800.0 PL=0
MOVL C01102 V=800.0 PL=0
MOVL C01103 V=800.0 PL=0
MOVL C01104 V=800.0 PL=0
MOVL C01105 V=800.0 PL=0
MOVL C01106 V=800.0 PL=0
MOVL C01107 V=800.0 PL=0
MOVL C01108 V=800.0 PL=0
MOVL C01109 V=800.0 PL=0
MOVL C01110 V=800.0 PL=0
MOVL C01111 V=800.0 PL=0
MOVL C01112 V=800.0 PL=0
MOVL C01113 V=800.0 PL=0
MOVL C01114 V=800.0 PL=0
MOVL C01115 V=800.0 PL=0
MOVL C01116 V=800.0 PL=0
MOVL C01117 V=800.0 PL=0
MOVL C01118 V=800.0 PL=0
MOVL C01119 V=800.0 PL=0
MOVL C01120 V=800.0 PL=0
MOVL C01121 V=800.0 PL=0
MOVL C01122 V=800.0 PL=0
MOVL C01123 V=800.0 PL=0
MOVL C01124 V=800.0 PL=0
MOVL C01125 V=800.0 PL=0
MOVL C01126 V=800.0 PL=0
MOVL C01127 V=800.0 PL=0
MOVL C01128 V=800.0 PL=0
MOVL C01129 V=800.0 PL=0
MOVL C01130 V=800.0 PL=0
MOVL C01131 V=800.0 PL=0
MOVL C01132 V=800.0 PL=0
MOVL C01133 V=800.0 PL=0
MOVL C01134 V=800.0 PL=0
MOVL C01135 V=800.0 PL=0
MOVL C01136 V=800.0 PL=0
MOVL C01137 V=800.0 PL=0
MOVL C01138 V=800.0 PL=0
MOVL C01139 V=800.0 PL=0
MOVL C01140 V=800.0 PL=0
MOVL C01141 V=800.0 PL=0
MOVL C01142 V=800.0 PL=0
MOVL C01143 V=800.0 PL=0
MOVL C01144 V=800.0 PL=0
MOVL C01145 V=800.0 PL=0
MOVL C01146 V=800.0 PL=0
MOVL C01147 V=800.0 PL=0
MOVL C01148 V=800.0 PL=0
MOVL C01149 V=800.0 PL=0
MOVL C01150 V=800.0 PL=0
MOVL C01151 V=800.0 PL=0
MOVL C01152 V=800.0 PL=0
MOVL C01153 V=800.0 PL=0
MOVL C01154 V=800.0 PL=0
MOVL C01155 V=800.0 PL=0
MOVL C01156 V=800.0 PL=0
MOVL C01157 V=800.0 PL=0
MOVL C01158 V=800.0 PL=0
MOVL C01159 V=800.0 PL=0
MOVL C01160 V=800.0 PL=0
MOVL C01161 V=800.0 PL=0
MOVL C01162 V=800.0 PL=0
MOVL C01163 V=800.0 PL=0
MOVL C01164 V=800.0 PL=0
MOVL C01165 V=800.0 PL=0
MOVL C01166 V=800.0 PL=0
MOVL C01167 V=800.0 PL=0
MOVL C01168 V=800.0 PL=0
MOVL C01169 V=800.0 PL=0
MOVL C01170 V=800.0 PL=0
MOVL C01171 V=800.0 PL=0
MOVL C01172 V=800.0 PL=0
MOVL C01173 V=800.0 PL=0
MOVL C01174 V=800.0 PL=0
MOVL C01175 V=800.0 PL=0
MOVL C01176 V=800.0 PL=0
MOVL C01177 V=800.0 PL=0
MOVL C01178 V=800.0 PL=0
MOVL C01179 V=800.0 PL=0
MOVL C01180 V=800.0 PL=0
MOVL C01181 V=800.0 PL=0
MOVL C01182 V=800.0 PL=0
MOVL C01183 V=800.0 PL=0
MOVL C01184 V=800.0 PL=0
MOVL C01185 V=800.0 PL=0
MOVL C01186 V=800.0 PL=0
MOVL C01187 V=800.0 PL=0
MOVL C01188 V=800.0 PL=0
MOVL C01189 V=800.0 PL=0
MOVL C01190 V=800.0 PL=0
MOVL C01191 V=800.0 PL=0
MOVL C01192 V=800.0 PL=0
MOVL C01193 V=800.0 PL=0
MOVL C01194 V=800.0 PL=0
MOVL C01195 V=800.0 PL=0
MOVL C01196 V=800.0 PL=0
MOVL C01197 V=800.0 PL=0
MOVL C01198 V=800.0 PL=0
MOVL C01199 V=800.0 PL=0
MOVL C01200 V=800.0 PL=0
MOVL C01201 V=800.0 PL=0
MOVL C01202 V=800.0 PL=0
MOVL C01203 V=800.0 PL=0
MOVL C01204 V=800.0 PL=0
MOVL C01205 V=800.0 PL=0
MOVL C01206 V=800.0 PL=0
MOVL C01207 V=800.0 PL=0
MOVL C01208 V=800.0 PL=0
MOVL C01209 V=800.0 PL=0
MOVL C01210 V=800.0 PL=0
MOVL C01211 V=800.0 PL=0
MOVL C01212 V=800.0 PL=0
MOVL C01213 V=800.0 PL=0
MOVL C01214 V=800.0 PL=0
MOVL C01215 V=800.0 PL=0
MOVL C01216 V=800.0 PL=0
MOVL C01217 V=800.0 PL=0
MOVL C01218 V=800.0 PL=0
MOVL C01219 V=800.0 PL=0
MOVL C01220 V=800.0 PL=0
MOVL C01221 V=800.0 PL=0
MOVL C01222 V=800.0 PL=0
MOVL C01223 V=800.0 PL=0
MOVL C01224 V=800.0 PL=0
MOVL C01225 V=800.0 PL=0
MOVL C01226 V=800.0 PL=0
MOVL C01227 V=800.0 PL=0
MOVL C01228 V=800.0 PL=0
MOVL C01229 V=800.0 PL=0
MOVL C01230 V=800.0 PL=0
MOVL C01231 V=800.0 PL=0
MOVL C01232 V=800.0 PL=0
MOVL C01233 V=800.0 PL=0
MOVL C01234 V=800.0 PL=0
MOVL C01235 V=800.0 PL=0
MOVL C01236 V=800.0 PL=0
MOVL C01237 V=800.0 PL=0
MOVL C01238 V=800.0 PL=0
MOVL C01239 V=800.0 PL=0
MOVL C01240 V=800.0 PL=0
MOVL C01241 V=800.0 PL=0
MOVL C01242 V=800.0 PL=0
MOVL C01243 V=800.0 PL=0
MOVL C01244 V=800.0 PL=0
MOVL C01245 V=800.0 PL=0
MOVL C01246 V=800.0 PL=0
MOVL C01247 V=800.0 PL=0
MOVL C01248 V=800.0 PL=0
MOVL C01249 V=800.0 PL=0
MOVL C01250 V=800.0 PL=0
MOVL C01251 V=800.0 PL=0
MOVL C01252 V=800.0 PL=0
MOVL C01253 V=800.0 PL=0
MOVL C01254 V=800.0 PL=0
MOVL C01255 V=800.0 PL=0
MOVL C01256 V=800.0 PL=0
MOVL C01257 V=800.0 PL=0
MOVL C01258 V=800.0 PL=0
MOVL C01259 V=800.0 PL=0
MOVL C01260 V=800.0 PL=0
MOVL C01261 V=800.0 PL=0
MOVL C01262 V=800.0 PL=0
MOVL C01263 V=800.0 PL=0
MOVL C01264 V=800.0 PL=0
MOVL C01265 V=800.0 PL=0
MOVL C01266 V=800.0 PL=0
MOVL C01267 V=800.0 PL=0
MOVL C01268 V=800.0 PL=0
MOVL C01269 V=800.0 PL=0
MOVL C01270 V=800.0 PL=0
MOVL C01271 V=800.0 PL=0
MOVL C01272 V=800.0 PL=0
MOVL C01273 V=800.0 PL=0
MOVL C01274 V=800.0 PL=0
MOVL C01275 V=800.0 PL=0
MOVL C01276 V=800.0 PL=0
MOVL C01277 V=800.0 PL=0
MOVL C01278 V=800.0 PL=0
MOVL C01279 V=800.0 PL=0
MOVL C01280 V=800.0 PL=0
MOVL C01281 V=800.0 PL=0
MOVL C01282 V=800.0 PL=0
MOVL C01283 V=800.0 PL=0
MOVL C01284 V=800.0 PL=0
MOVL C01285 V=800.0 PL=0
MOVL C01286 V=800.0 PL=0
MOVL C01287 V=800.0 PL=0
MOVL C01288 V=800.0 PL=0
MOVL C01289 V=800.0 PL=0
MOVL C01290 V=800.0 PL=0
MOVL C01291 V=800.0 PL=0
MOVL C01292 V=800.0 PL=0
MOVL C01293 V=800.0 PL=0
MOVL C01294 V=800.0 PL=0
MOVL C01295 V=800.0 PL=0
MOVL C01296 V=800.0 PL=0
MOVL C01297 V=800.0 PL=0
MOVL C01298 V=800.0 PL=0
MOVL C01299 V=800.0 PL=0
MOVL C01300 V=800.0 PL=0
MOVL C01301 V=800.0 PL=0
MOVL C01302 V=800.0 PL=0
MOVL C01303 V=800.0 PL=0
MOVL C01304 V=800.0 PL=0
MOVL C01305 V=800.0 PL=0
MOVL C01306 V=800.0 PL=0
MOVL C01307 V=800.0 PL=0
MOVL C01308 V=800.0 PL=0
MOVL C01309 V=800.0 PL=0
MOVL C01310 V=800.0 PL=0
MOVL C01311 V=800.0 PL=0
MOVL C01312 V=800.0 PL=0
MOVL C01313 V=800.0 PL=0
MOVL C01314 V=800.0 PL=0
MOVL C01315 V=800.0 PL=0
MOVL C01316 V=800.0 PL=0
MOVL C01317 V=800.0 PL=0
MOVL C01318 V=800.0 PL=0
MOVL C01319 V=800.0 PL=0
MOVL C01320 V=800.0 PL=0
MOVL C01321 V=800.0 PL=0
MOVL C01322 V=800.0 PL=0
MOVL C01323 V=800.0 PL=0
MOVL C01324 V=800.0 PL=0
MOVL C01325 V=800.0 PL=0
MOVL C01326 V=800.0 PL=0
MOVL C01327 V=800.0 PL=0
MOVL C01328 V=800.0 PL=0
MOVL C01329 V=800.0 PL=0
MOVL C01330 V=800.0 PL=0
MOVL C01331 V=800.0 PL=0
MOVL C01332 V=800.0 PL=0
MOVL C01333 V=800.0 PL=0
MOVL C01334 V=800.0 PL=0
MOVL C01335 V=800.0 PL=0
MOVL C01336 V=800.0 PL=0
MOVL C01337 V=800.0 PL=0
MOVL C01338 V=800.0 PL=0
MOVL C01339 V=800.0 PL=0
MOVL C01340 V=800.0 PL=0
MOVL C01341 V=800.0 PL=0
MOVL C01342 V=800.0 PL=0
MOVL C01343 V=800.0 PL=0
MOVL C01344 V=800.0 PL=0
MOVL C01345 V=800.0 PL=0
MOVL C01346 V=800.0 PL=0
MOVL C01347 V=800.0 PL=0
MOVL C01348 V=800.0 PL=0
MOVL C01349 V=800.0 PL=0
MOVL C01350 V=800.0 PL=0
MOVL C01351 V=800.0 PL=0
MOVL C01352 V=800.0 PL=0
MOVL C01353 V=800.0 PL=0
MOVL C01354 V=800.0 PL=0
MOVL C01355 V=800.0 PL=0
MOVL C01356 V=800.0 PL=0
MOVL C01357 V=800.0 PL=0
MOVL C01358 V=800.0 PL=0
MOVL C01359 V=800.0 PL=0
MOVL C01360 V=800.0 PL=0
MOVL C01361 V=800.0 PL=0
MOVL C01362 V=800.0 PL=0
MOVL C01363 V=800.0 PL=0
MOVL C01364 V=800.0 PL=0
MOVL C01365 V=800.0 PL=0
MOVL C01366 V=800.0 PL=0
MOVL C01367 V=800.0 PL=0
MOVL C01368 V=800.0 PL=0
MOVL C01369 V=800.0 PL=0
MOVL C01370 V=800.0 PL=0
MOVL C01371 V=800.0 PL=0
MOVL C01372 V=800.0 PL=0
MOVL C01373 V=800.0 PL=0
MOVL C01374 V=800.0 PL=0
MOVL C01375 V=800.0 PL=0
MOVL C01376 V=800.0 PL=0
MOVL C01377 V=800.0 PL=0
MOVL C01378 V=800.0 PL=0
MOVL C01379 V=800.0 PL=0
MOVL C01380 V=800.0 PL=0
MOVL C01381 V=800.0 PL=0
MOVL C01382 V=800.0 PL=0
MOVL C01383 V=800.0 PL=0
MOVL C01384 V=800.0 PL=0
MOVL C01385 V=800.0 PL=0
MOVL C01386 V=800.0 PL=0
MOVL C01387 V=800.0 PL=0
MOVL C01388 V=800.0 PL=0
MOVL C01389 V=800.0 PL=0
MOVL C01390 V=800.0 PL=0
MOVL C01391 V=800.0 PL=0
MOVL C01392 V=800.0 PL=0
MOVL C01393 V=800.0 PL=0
MOVL C01394 V=800.0 PL=0
MOVL C01395 V=800.0 PL=0
MOVL C01396 V=800.0 PL=0
MOVL C01397 V=800.0 PL=0
MOVL C01398 V=800.0 PL=0
MOVL C01399 V=800.0 PL=0
MOVL C01400 V=800.0 PL=0
MOVL C01401 V=800.0 PL=0
MOVL C01402 V=800.0 PL=0
MOVL C01403 V=800.0 PL=0
MOVL C01404 V=800.0 PL=0
MOVL C01405 V=800.0 PL=0
MOVL C01406 V=800.0 PL=0
MOVL C01407 V=800.0 PL=0
MOVL C01408 V=800.0 PL=0
MOVL C01409 V=800.0 PL=0
MOVL C01410 V=800.0 PL=0
MOVL C01411 V=800.0 PL=0
MOVL C01412 V=800.0 PL=0
MOVL C01413 V=800.0 PL=0
MOVL C01414 V=800.0 PL=0
MOVL C01415 V=800.0 PL=0
MOVL C01416 V=800.0 PL=0
MOVL C01417 V=800.0 PL=0
MOVL C01418 V=800.0 PL=0
MOVL C01419 V=800.0 PL=0
MOVL C01420 V=800.0 PL=0
MOVL C01421 V=800.0 PL=0
MOVL C01422 V=800.0 PL=0
MOVL C01423 V=800.0 PL=0
MOVL C01424 V=800.0 PL=0
MOVL C01425 V=800.0 PL=0
MOVL C01426 V=800.0 PL=0
MOVL C01427 V=800.0 PL=0
MOVL C01428 V=800.0 PL=0
MOVL C01429 V=800.0 PL=0
MOVL C01430 V=800.0 PL=0
MOVL C01431 V=800.0 PL=0
MOVL C01432 V=800.0 PL=0
MOVL C01433 V=800.0 PL=0
MOVL C01434 V=800.0 PL=0
MOVL C01435 V=800.0 PL=0
MOVL C01436 V=800.0 PL=0
MOVL C01437 V=800.0 PL=0
MOVL C01438 V=800.0 PL=0
MOVL C01439 V=800.0 PL=0
MOVL C01440 V=800.0 PL=0
MOVL C01441 V=800.0 PL=0
MOVL C01442 V=800.0 PL=0
MOVL C01443 V=800.0 PL=0
MOVL C01444 V=800.0 PL=0
MOVL C01445 V=800.0 PL=0
MOVL C01446 V=800.0 PL=0
MOVL C01447 V=800.0 PL=0
MOVL C01448 V=800.0 PL=0
MOVL C01449 V=800.0 PL=0
MOVL C01450 V=800.0 PL=0
MOVL C01451 V=800.0 PL=0
MOVL C01452 V=800.0 PL=0
MOVL C01453 V=800.0 PL=0
MOVL C01454 V=800.0 PL=0
MOVL C01455 V=800.0 PL=0
MOVL C01456 V=800.0 PL=0
MOVL C01457 V=800.0 PL=0
MOVL C01458 V=800.0 PL=0
MOVL C01459 V=800.0 PL=0
MOVL C01460 V=800.0 PL=0
MOVL C01461 V=800.0 PL=0
MOVL C01462 V=800.0 PL=0
MOVL C01463 V=800.0 PL=0
MOVL C01464 V=800.0 PL=0
MOVL C01465 V=800.0 PL=0
MOVL C01466 V=800.0 PL=0
MOVL C01467 V=800.0 PL=0
MOVL C01468 V=800.0 PL=0
MOVL C01469 V=800.0 PL=0
MOVL C01470 V=800.0 PL=0
MOVL C01471 V=800.0 PL=0
MOVL C01472 V=800.0 PL=0
MOVL C01473 V=800.0 PL=0
MOVL C01474 V=800.0 PL=0
MOVL C01475 V=800.0 PL=0
MOVL C01476 V=800.0 PL=0
MOVL C01477 V=800.0 PL=0
MOVL C01478 V=800.0 PL=0
MOVL C01479 V=800.0 PL=0
MOVL C01480 V=800.0 PL=0
MOVL C01481 V=800.0 PL=0
MOVL C01482 V=800.0 PL=0
MOVL C01483 V=800.0 PL=0
MOVL C01484 V=800.0 PL=0
MOVL C01485 V=800.0 PL=0
MOVL C01486 V=800.0 PL=0
MOVL C01487 V=800.0 PL=0
MOVL C01488 V=800.0 PL=0
MOVL C01489 V=800.0 PL=0
MOVL C01490 V=800.0 PL=0
MOVL C01491 V=800.0 PL=0
MOVL C01492 V=800.0 PL=0
MOVL C01493 V=800.0 PL=0
MOVL C01494 V=800.0 PL=0
MOVL C01495 V=800.0 PL=0
MOVL C01496 V=800.0 PL=0
MOVL C01497 V=800.0 PL=0
MOVL C01498 V=800.0 PL=0
MOVL C01499 V=800.0 PL=0
MOVL C01500 V=800.0 PL=0
MOVL C01501 V=800.0 PL=0
MOVL C01502 V=800.0 PL=0
MOVL C01503 V=800.0 PL=0
MOVL C01504 V=800.0 PL=0
MOVL C01505 V=800.0 PL=0
MOVL C01506 V=800.0 PL=0
MOVL C01507 V=800.0 PL=0
MOVL C01508 V=800.0 PL=0
MOVL C01509 V=800.0 PL=0
MOVL C01510 V=800.0 PL=0
MOVL C01511 V=800.0 PL=0
MOVL C01512 V=800.0 PL=0
MOVL C01513 V=800.0 PL=0
MOVL C01514 V=800.0 PL=0
MOVL C01515 V=800.0 PL=0
MOVL C01516 V=800.0 PL=0
MOVL C01517 V=800.0 PL=0
MOVL C01518 V=800.0 PL=0
MOVL C01519 V=800.0 PL=0
MOVL C01520 V=800.0 PL=0
MOVL C01521 V=800.0 PL=0
MOVL C01522 V=800.0 PL=0
MOVL C01523 V=800.0 PL=0
MOVL C01524 V=800.0 PL=0
MOVL C01525 V=800.0 PL=0
MOVL C01526 V=800.0 PL=0
MOVL C01527 V=800.0 PL=0
MOVL C01528 V=800.0 PL=0
MOVL C01529 V=800.0 PL=0
MOVL C01530 V=800.0 PL=0
MOVL C01531 V=800.0 PL=0
MOVL C01532 V=800.0 PL=0
MOVL C01533 V=800.0 PL=0
MOVL C01534 V=800.0 PL=0
MOVL C01535 V=800.0 PL=0
MOVL C01536 V=800.0 PL=0
MOVL C01537 V=800.0 PL=0
MOVL C01538 V=800.0 PL=0
MOVL C01539 V=800.0 PL=0
MOVL C01540 V=800.0 PL=0
MOVL C01541 V=800.0 PL=0
MOVL C01542 V=800.0 PL=0
MOVL C01543 V=800.0 PL=0
MOVL C01544 V=800.0 PL=0
MOVL C01545 V=800.0 PL=0
MOVL C01546 V=800.0 PL=0
MOVL C01547 V=800.0 PL=0
MOVL C01548 V=800.0 PL=0
MOVL C01549 V=800.0 PL=0
MOVL C01550 V=800.0 PL=0
MOVL C01551 V=800.0 PL=0
MOVL C01552 V=800.0 PL=0
MOVL C01553 V=800.0 PL=0
MOVL C01554 V=800.0 PL=0
MOVL C01555 V=800.0 PL=0
MOVL C01556 V=800.0 PL=0
MOVL C01557 V=800.0 PL=0
MOVL C01558 V=800.0 PL=0
MOVL C01559 V=800.0 PL=0
MOVL C01560 V=800.0 PL=0
MOVL C01561 V=800.0 PL=0
MOVL C01562 V=800.0 PL=0
MOVL C01563 V=800.0 PL=0
MOVL C01564 V=800.0 PL=0
MOVL C01565 V=800.0 PL=0
MOVL C01566 V=800.0 PL=0
MOVL C01567 V=800.0 PL=0
MOVL C01568 V=800.0 PL=0
MOVL C01569 V=800.0 PL=0
MOVL C01570 V=800.0 PL=0
MOVL C01571 V=800.0 PL=0
MOVL C01572 V=800.0 PL=0
MOVL C01573 V=800.0 PL=0
MOVL C01574 V=800.0 PL=0
MOVL C01575 V=800.0 PL=0
MOVL C01576 V=800.0 PL=0
MOVL C01577 V=800.0 PL=0
MOVL C01578 V=800.0 PL=0
MOVL C01579 V=800.0 PL=0
MOVL C01580 V=800.0 PL=0
MOVL C01581 V=800.0 PL=0
MOVL C01582 V=800.0 PL=0
MOVL C01583 V=800.0 PL=0
MOVL C01584 V=800.0 PL=0
MOVL C01585 V=800.0 PL=0
MOVL C01586 V=800.0 PL=0
MOVL C01587 V=800.0 PL=0
MOVL C01588 V=800.0 PL=0
MOVL C01589 V=800.0 PL=0
MOVL C01590 V=800.0 PL=0
MOVL C01591 V=800.0 PL=0
MOVL C01592 V=800.0 PL=0
MOVL C01593 V=800.0 PL=0
MOVL C01594 V=800.0 PL=0
MOVL C01595 V=800.0 PL=0
MOVL C01596 V=800.0 PL=0
MOVL C01597 V=800.0 PL=0
MOVL C01598 V=800.0 PL=0
MOVL C01599 V=800.0 PL=0
MOVL C01600 V=800.0 PL=0
MOVL C01601 V=800.0 PL=0
MOVL C01602 V=800.0 PL=0
MOVL C01603 V=800.0 PL=0
MOVL C01604 V=800.0 PL=0
MOVL C01605 V=800.0 PL=0
MOVL C01606 V=800.0 PL=0
MOVL C01607 V=800.0 PL=0
MOVL C01608 V=800.0 PL=0
MOVL C01609 V=800.0 PL=0
MOVL C01610 V=800.0 PL=0
MOVL C01611 V=800.0 PL=0
MOVL C01612 V=800.0 PL=0
MOVL C01613 V=800.0 PL=0
MOVL C01614 V=800.0 PL=0
MOVL C01615 V=800.0 PL=0
MOVL C01616 V=800.0 PL=0
MOVL C01617 V=800.0 PL=0
MOVL C01618 V=800.0 PL=0
MOVL C01619 V=800.0 PL=0
MOVL C01620 V=800.0 PL=0
MOVL C01621 V=800.0 PL=0
MOVL C01622 V=800.0 PL=0
MOVL C01623 V=800.0 PL=0
MOVL C01624 V=800.0 PL=0
MOVL C01625 V=800.0 PL=0
MOVL C01626 V=800.0 PL=0
MOVL C01627 V=800.0 PL=0
MOVL C01628 V=800.0 PL=0
MOVL C01629 V=800.0 PL=0
MOVL C01630 V=800.0 PL=0
MOVL C01631 V=800.0 PL=0
MOVL C01632 V=800.0 PL=0
MOVL C01633 V=800.0 PL=0
MOVL C01634 V=800.0 PL=0
MOVL C01635 V=800.0 PL=0
MOVL C01636 V=800.0 PL=0
MOVL C01637 V=800.0 PL=0
MOVL C01638 V=800.0 PL=0
MOVL C01639 V=800.0 PL=0
MOVL C01640 V=800.0 PL=0
MOVL C01641 V=800.0 PL=0
MOVL C01642 V=800.0 PL=0
MOVL C01643 V=800.0 PL=0
MOVL C01644 V=800.0 PL=0
MOVL C01645 V=800.0 PL=0
MOVL C01646 V=800.0 PL=0
MOVL C01647 V=800.0 PL=0
MOVL C01648 V=800.0 PL=0
MOVL C01649 V=800.0 PL=0
MOVL C01650 V=800.0 PL=0
MOVL C01651 V=800.0 PL=0
MOVL C01652 V=800.0 PL=0
MOVL C01653 V=800.0 PL=0
MOVL C01654 V=800.0 PL=0
MOVL C01655 V=800.0 PL=0
MOVL C01656 V=800.0 PL=0
MOVL C01657 V=800.0 PL=0
MOVL C01658 V=800.0 PL=0
MOVL C01659 V=800.0 PL=0
MOVL C01660 V=800.0 PL=0
MOVL C01661 V=800.0 PL=0
MOVL C01662 V=800.0 PL=0
MOVL C01663 V=800.0 PL=0
MOVL C01664 V=800.0 PL=0
MOVL C01665 V=800.0 PL=0
MOVL C01666 V=800.0 PL=0
MOVL C01667 V=800.0 PL=0
MOVL C01668 V=800.0 PL=0
MOVL C01669 V=800.0 PL=0
MOVL C01670 V=800.0 PL=0
MOVL C01671 V=800.0 PL=0
MOVL C01672 V=800.0 PL=0
MOVL C01673 V=800.0 PL=0
MOVL C01674 V=800.0 PL=0
MOVL C01675 V=800.0 PL=0
MOVL C01676 V=800.0 PL=0
MOVL C01677 V=800.0 PL=0
MOVL C01678 V=800.0 PL=0
MOVL C01679 V=800.0 PL=0
MOVL C01680 V=800.0 PL=0
MOVL C01681 V=800.0 PL=0
MOVL C01682 V=800.0 PL=0
MOVL C01683 V=800.0 PL=0
MOVL C01684 V=800.0 PL=0
MOVL C01685 V=800.0 PL=0
MOVL C01686 V=800.0 PL=0
MOVL C01687 V=800.0 PL=0
MOVL C01688 V=800.0 PL=0
MOVL C01689 V=800.0 PL=0
MOVL C01690 V=800.0 PL=0
MOVL C01691 V=800.0 PL=0
MOVL C01692 V=800.0 PL=0
MOVL C01693 V=800.0 PL=0
MOVL C01694 V=800.0 PL=0
MOVL C01695 V=800.0 PL=0
MOVL C01696 V=800.0 PL=0
MOVL C01697 V=800.0 PL=0
MOVL C01698 V=800.0 PL=0
MOVL C01699 V=800.0 PL=0
MOVL C01700 V=800.0 PL=0
MOVL C01701 V=800.0 PL=0
MOVL C01702 V=800.0 PL=0
MOVL C01703 V=800.0 PL=0
MOVL C01704 V=800.0 PL=0
MOVL C01705 V=800.0 PL=0
MOVL C01706 V=800.0 PL=0
MOVL C01707 V=800.0 PL=0
MOVL C01708 V=800.0 PL=0
MOVL C01709 V=800.0 PL=0
MOVL C01710 V=800.0 PL=0
MOVL C01711 V=800.0 PL=0
MOVL C01712 V=800.0 PL=0
MOVL C01713 V=800.0 PL=0
MOVL C01714 V=800.0 PL=0
MOVL C01715 V=800.0 PL=0
MOVL C01716 V=800.0 PL=0
MOVL C01717 V=800.0 PL=0
MOVL C01718 V=800.0 PL=0
MOVL C01719 V=800.0 PL=0
MOVL C01720 V=800.0 PL=0
MOVL C01721 V=800.0 PL=0
MOVL C01722 V=800.0 PL=0
MOVL C01723 V=800.0 PL=0
MOVL C01724 V=800.0 PL=0
MOVL C01725 V=800.0 PL=0
MOVL C01726 V=800.0 PL=0
MOVL C01727 V=800.0 PL=0
MOVL C01728 V=800.0 PL=0
MOVL C01729 V=800.0 PL=0
MOVL C01730 V=800.0 PL=0
MOVL C01731 V=800.0 PL=0
MOVL C01732 V=800.0 PL=0
MOVL C01733 V=800.0 PL=0
MOVL C01734 V=800.0 PL=0
MOVL C01735 V=800.0 PL=0
MOVL C01736 V=800.0 PL=0
MOVL C01737 V=800.0 PL=0
MOVL C01738 V=800.0 PL=0
MOVL C01739 V=800.0 PL=0
MOVL C01740 V=800.0 PL=0
MOVL C01741 V=800.0 PL=0
MOVL C01742 V=800.0 PL=0
MOVL C01743 V=800.0 PL=0
MOVL C01744 V=800.0 PL=0
MOVL C01745 V=800.0 PL=0
MOVL C01746 V=800.0 PL=0
MOVL C01747 V=800.0 PL=0
MOVL C01748 V=800.0 PL=0
MOVL C01749 V=800.0 PL=0
MOVL C01750 V=800.0 PL=0
MOVL C01751 V=800.0 PL=0
MOVL C01752 V=800.0 PL=0
MOVL C01753 V=800.0 PL=0
MOVL C01754 V=800.0 PL=0
MOVL C01755 V=800.0 PL=0
MOVL C01756 V=800.0 PL=0
MOVL C01757 V=800.0 PL=0
MOVL C01758 V=800.0 PL=0
MOVL C01759 V=800.0 PL=0
MOVL C01760 V=800.0 PL=0
MOVL C01761 V=800.0 PL=0
MOVL C01762 V=800.0 PL=0
MOVL C01763 V=800.0 PL=0
MOVL C01764 V=800.0 PL=0
MOVL C01765 V=800.0 PL=0
MOVL C01766 V=800.0 PL=0
MOVL C01767 V=800.0 PL=0
MOVL C01768 V=800.0 PL=0
MOVL C01769 V=800.0 PL=0
MOVL C01770 V=800.0 PL=0
MOVL C01771 V=800.0 PL=0
MOVL C01772 V=800.0 PL=0
MOVL C01773 V=800.0 PL=0
MOVL C01774 V=800.0 PL=0
MOVL C01775 V=800.0 PL=0
MOVL C01776 V=800.0 PL=0
MOVL C01777 V=800.0 PL=0
MOVL C01778 V=800.0 PL=0
MOVL C01779 V=800.0 PL=0
MOVL C01780 V=800.0 PL=0
MOVL C01781 V=800.0 PL=0
MOVL C01782 V=800.0 PL=0
MOVL C01783 V=800.0 PL=0
MOVL C01784 V=800.0 PL=0
MOVL C01785 V=800.0 PL=0
MOVL C01786 V=800.0 PL=0
MOVL C01787 V=800.0 PL=0
MOVL C01788 V=800.0 PL=0
MOVL C01789 V=800.0 PL=0
MOVL C01790 V=800.0 PL=0
MOVL C01791 V=800.0 PL=0
MOVL C01792 V=800.0 PL=0
MOVL C01793 V=800.0 PL=0
MOVL C01794 V=800.0 PL=0
MOVL C01795 V=800.0 PL=0
MOVL C01796 V=800.0 PL=0
MOVL C01797 V=800.0 PL=0
MOVL C01798 V=800.0 PL=0
MOVL C01799 V=800.0 PL=0
MOVL C01800 V=800.0 PL=0
MOVL C01801 V=800.0 PL=0
MOVL C01802 V=800.0 PL=0
MOVL C01803 V=800.0 PL=0
MOVL C01804 V=800.0 PL=0
MOVL C01805 V=800.0 PL=0
MOVL C01806 V=800.0 PL=0
MOVL C01807 V=800.0 PL=0
MOVL C01808 V=800.0 PL=0
MOVL C01809 V=800.0 PL=0
MOVL C01810 V=800.0 PL=0
MOVL C01811 V=800.0 PL=0
MOVL C01812 V=800.0 PL=0
MOVL C01813 V=800.0 PL=0
MOVL C01814 V=800.0 PL=0
MOVL C01815 V=800.0 PL=0
MOVL C01816 V=800.0 PL=0
MOVL C01817 V=800.0 PL=0
MOVL C01818 V=800.0 PL=0
MOVL C01819 V=800.0 PL=0
MOVL C01820 V=800.0 PL=0
MOVL C01821 V=800.0 PL=0
MOVL C01822 V=800.0 PL=0
MOVL C01823 V=800.0 PL=0
MOVL C01824 V=800.0 PL=0
MOVL C01825 V=800.0 PL=0
MOVL C01826 V=800.0 PL=0
MOVL C01827 V=800.0 PL=0
MOVL C01828 V=800.0 PL=0
MOVL C01829 V=800.0 PL=0
MOVL C01830 V=800.0 PL=0
MOVL C01831 V=800.0 PL=0
MOVL C01832 V=800.0 PL=0
MOVL C01833 V=800.0 PL=0
MOVL C01834 V=800.0 PL=0
MOVL C01835 V=800.0 PL=0
MOVL C01836 V=800.0 PL=0
MOVL C01837 V=800.0 PL=0
MOVL C01838 V=800.0 PL=0
MOVL C01839 V=800.0 PL=0
MOVL C01840 V=800.0 PL=0
MOVL C01841 V=800.0 PL=0
MOVL C01842 V=800.0 PL=0
MOVL C01843 V=800.0 PL=0
MOVL C01844 V=800.0 PL=0
MOVL C01845 V=800.0 PL=0
MOVL C01846 V=800.0 PL=0
MOVL C01847 V=800.0 PL=0
MOVL C01848 V=800.0 PL=0
MOVL C01849 V=800.0 PL=0
MOVL C01850 V=800.0 PL=0
MOVL C01851 V=800.0 PL=0
MOVL C01852 V=800.0 PL=0
MOVL C01853 V=800.0 PL=0
MOVL C01854 V=800.0 PL=0
MOVL C01855 V=800.0 PL=0
MOVL C01856 V=800.0 PL=0
MOVL C01857 V=800.0 PL=0
MOVL C01858 V=800.0 PL=0
MOVL C01859 V=800.0 PL=0
MOVL C01860 V=800.0 PL=0
MOVL C01861 V=800.0 PL=0
MOVL C01862 V=800.0 PL=0
MOVL C01863 V=800.0 PL=0
MOVL C01864 V=800.0 PL=0
MOVL C01865 V=800.0 PL=0
MOVL C01866 V=800.0 PL=0
MOVL C01867 V=800.0 PL=0
MOVL C01868 V=800.0 PL=0
MOVL C01869 V=800.0 PL=0
MOVL C01870 V=800.0 PL=0
MOVL C01871 V=800.0 PL=0
MOVL C01872 V=800.0 PL=0
MOVL C01873 V=800.0 PL=0
MOVL C01874 V=800.0 PL=0
MOVL C01875 V=800.0 PL=0
MOVL C01876 V=800.0 PL=0
MOVL C01877 V=800.0 PL=0
MOVL C01878 V=800.0 PL=0
MOVL C01879 V=800.0 PL=0
MOVL C01880 V=800.0 PL=0
MOVL C01881 V=800.0 PL=0
MOVL C01882 V=800.0 PL=0
MOVL C01883 V=800.0 PL=0
MOVL C01884 V=800.0 PL=0
MOVL C01885 V=800.0 PL=0
MOVL C01886 V=800.0 PL=0
MOVL C01887 V=800.0 PL=0
MOVL C01888 V=800.0 PL=0
MOVL C01889 V=800.0 PL=0
MOVL C01890 V=800.0 PL=0
MOVL C01891 V=800.0 PL=0
MOVL C01892 V=800.0 PL=0
MOVL C01893 V=800.0 PL=0
MOVL C01894 V=800.0 PL=0
MOVL C01895 V=800.0 PL=0
MOVL C01896 V=800.0 PL=0
MOVL C01897 V=800.0 PL=0
MOVL C01898 V=800.0 PL=0
MOVL C01899 V=800.0 PL=0
MOVL C01900 V=800.0 PL=0
MOVL C01901 V=800.0 PL=0
MOVL C01902 V=800.0 PL=0
MOVL C01903 V=800.0 PL=0
MOVL C01904 V=800.0 PL=0
MOVL C01905 V=800.0 PL=0
MOVL C01906 V=800.0 PL=0
MOVL C01907 V=800.0 PL=0
MOVL C01908 V=800.0 PL=0
MOVL C01909 V=800.0 PL=0
MOVL C01910 V=800.0 PL=0
MOVL C01911 V=800.0 PL=0
MOVL C01912 V=800.0 PL=0
MOVL C01913 V=800.0 PL=0
MOVL C01914 V=800.0 PL=0
MOVL C01915 V=800.0 PL=0
MOVL C01916 V=800.0 PL=0
MOVL C01917 V=800.0 PL=0
MOVL C01918 V=800.0 PL=0
MOVL C01919 V=800.0 PL=0
MOVL C01920 V=800.0 PL=0
MOVL C01921 V=800.0 PL=0
MOVL C01922 V=800.0 PL=0
MOVL C01923 V=800.0 PL=0
MOVL C01924 V=800.0 PL=0
MOVL C01925 V=800.0 PL=0
MOVL C01926 V=800.0 PL=0
MOVL C01927 V=800.0 PL=0
MOVL C01928 V=800.0 PL=0
MOVL C01929 V=800.0 PL=0
MOVL C01930 V=800.0 PL=0
MOVL C01931 V=800.0 PL=0
MOVL C01932 V=800.0 PL=0
MOVL C01933 V=800.0 PL=0
MOVL C01934 V=800.0 PL=0
MOVL C01935 V=800.0 PL=0
MOVL C01936 V=800.0 PL=0
MOVL C01937 V=800.0 PL=0
MOVL C01938 V=800.0 PL=0
MOVL C01939 V=800.0 PL=0
MOVL C01940 V=800.0 PL=0
MOVL C01941 V=800.0 PL=0
MOVL C01942 V=800.0 PL=0
MOVL C01943 V=800.0 PL=0
MOVL C01944 V=800.0 PL=0
MOVL C01945 V=800.0 PL=0
MOVL C01946 V=800.0 PL=0
MOVL C01947 V=800.0 PL=0
MOVL C01948 V=800.0 PL=0
MOVL C01949 V=800.0 PL=0
MOVL C01950 V=800.0 PL=0
MOVL C01951 V=800.0 PL=0
MOVL C01952 V=800.0 PL=0
MOVL C01953 V=800.0 PL=0
MOVL C01954 V=800.0 PL=0
MOVL C01955 V=800.0 PL=0
MOVL C01956 V=800.0 PL=0
MOVL C01957 V=800.0 PL=0
MOVL C01958 V=800.0 PL=0
MOVL C01959 V=800.0 PL=0
MOVL C01960 V=800.0 PL=0
MOVL C01961 V=800.0 PL=0
MOVL C01962 V=800.0 PL=0
MOVL C01963 V=800.0 PL=0
MOVL C01964 V=800.0 PL=0
MOVL C01965 V=800.0 PL=0
MOVL C01966 V=800.0 PL=0
MOVL C01967 V=800.0 PL=0
MOVL C01968 V=800.0 PL=0
MOVL C01969 V=800.0 PL=0
MOVL C01970 V=800.0 PL=0
MOVL C01971 V=800.0 PL=0
MOVL C01972 V=800.0 PL=0
MOVL C01973 V=800.0 PL=0
MOVL C01974 V=800.0 PL=0
MOVL C01975 V=800.0 PL=0
MOVL C01976 V=800.0 PL=0
MOVL C01977 V=800.0 PL=0
MOVL C01978 V=800.0 PL=0
MOVL C01979 V=800.0 PL=0
MOVL C01980 V=800.0 PL=0
MOVL C01981 V=800.0 PL=0
MOVL C01982 V=800.0 PL=0
MOVL C01983 V=800.0 PL=0
MOVL C01984 V=800.0 PL=0
MOVL C01985 V=800.0 PL=0
MOVL C01986 V=800.0 PL=0
MOVL C01987 V=800.0 PL=0
MOVL C01988 V=800.0 PL=0
MOVL C01989 V=800.0 PL=0
MOVL C01990 V=800.0 PL=0
MOVL C01991 V=800.0 PL=0
MOVL C01992 V=800.0 PL=0
MOVL C01993 V=800.0 PL=0
MOVL C01994 V=800.0 PL=0
MOVL C01995 V=800.0 PL=0
MOVL C01996 V=800.0 PL=0
MOVL C01997 V=800.0 PL=0
MOVL C01998 V=800.0 PL=0
MOVL C01999 V=800.0 PL=0
MOVL C02000 V=800.0 PL=0
MOVL C02001 V=800.0 PL=0
MOVL C02002 V=800.0 PL=0
MOVL C02003 V=800.0 PL=0
MOVL C02004 V=800.0 PL=0
MOVL C02005 V=800.0 PL=0
MOVL C02006 V=800.0 PL=0
MOVL C02007 V=800.0 PL=0
